LIN {X 0,Y 418.051,Z 411.422,A -85,B 0,C 180,E1 -10031.276,E2 -10031.276} C_VEL
LIN {X 0,Y 417.717,Z 417.579,A -85,B 0,C 180,E1 -10032.621,E2 -10032.621} C_VEL
LIN {X 0,Y 417.509,Z 421.319,A -85,B 0,C 180,E1 -10033.641,E2 -10033.641} C_VEL
LIN {X 0,Y 417.431,Z 423.461,A -85,B 0,C 180,E1 -10034.319,E2 -10034.319} C_VEL
LIN {X 0,Y 417.246,Z 426.661,A -85,B 0,C 180,E1 -10035.665,E2 -10035.665} C_VEL
LIN {X 0,Y 417.136,Z 427.966,A -85,B 0,C 180,E1 -10036.424,E2 -10036.424} C_VEL
LIN {X 0,Y 417.036,Z 429.647,A -85,B 0,C 180,E1 -10037.858,E2 -10037.858} C_VEL
LIN {X 0,Y 417.046,Z 430.141,A -85,B 0,C 180,E1 -10039.316,E2 -10039.316} C_VEL
LIN {X 0,Y 417.093,Z 429.416,A -85,B 0,C 180,E1 -10040.812,E2 -10040.812} C_VEL
LIN {X 0,Y 417.157,Z 428.808,A -85,B 0,C 180,E1 -10041.44,E2 -10041.44} C_VEL
LIN {X 0,Y 417.345,Z 426.876,A -85,B 0,C 180,E1 -10042.684,E2 -10042.684} C_VEL
LIN {X 0,Y 417.561,Z 424.076,A -85,B 0,C 180,E1 -10043.909,E2 -10043.909} C_VEL
LIN {X 0,Y 417.79,Z 420.364,A -85,B 0,C 180,E1 -10045.116,E2 -10045.116} C_VEL
LIN {X 0,Y 418.154,Z 414.507,A -85,B 0,C 180,E1 -10046.541,E2 -10046.541} C_VEL
LIN {X 0,Y 418.405,Z 409.706,A -85,B 0,C 180,E1 -10047.487,E2 -10047.487} C_VEL
LIN {X 0,Y 418.786,Z 403.362,A -85,B 0,C 180,E1 -10048.512,E2 -10048.512} C_VEL
LIN {X 0,Y 419.241,Z 396.766,A -85,B 0,C 180,E1 -10049.391,E2 -10049.391} C_VEL
LIN {X 0,Y 419.666,Z 389.265,A -85,B 0,C 180,E1 -10050.218,E2 -10050.218} C_VEL
LIN {X 0,Y 420.012,Z 381.871,A -85,B 0,C 180,E1 -10050.89,E2 -10050.89} C_VEL
LIN {X 0,Y 420.306,Z 374.017,A -85,B 0,C 180,E1 -10051.473,E2 -10051.473} C_VEL
LIN {X 0,Y 420.619,Z 365.492,A -85,B 0,C 180,E1 -10051.971,E2 -10051.971} C_VEL
LIN {X 0,Y 420.835,Z 356.386,A -85,B 0,C 180,E1 -10052.372,E2 -10052.372} C_VEL
LIN {X 0,Y 420.988,Z 346.253,A -85,B 0,C 180,E1 -10052.673,E2 -10052.673} C_VEL
LIN {X 0,Y 421.787,Z 285.672,A -85,B 0,C 180,E1 -10053.798,E2 -10053.798} C_VEL
LIN {X 0,Y 418.899,Z 271.189,A -85,B 0,C 180,E1 -10054.204,E2 -10054.204} C_VEL
LIN {X 0,Y 418.714,Z 265.669,A -85,B 0,C 180,E1 -10055.455,E2 -10055.455} C_VEL
LIN {X 0,Y 418.251,Z 263.201,A -85,B 0,C 180,E1 -10056.086,E2 -10056.086} C_VEL
LIN {X 0,Y 418.238,Z 263.204,A -85,B 0,C 180,E1 -10059.338,E2 -10059.338} C_VEL
LIN {X 0,Y 418.277,Z 263.2,A -85,B 0,C 180,E1 -10062.397,E2 -10062.397} C_VEL
LIN {X 0,Y 418.292,Z 263.192,A -85,B 0,C 180,E1 -10065.404,E2 -10065.404} C_VEL
LIN {X 0,Y 418.307,Z 263.193,A -85,B 0,C 180,E1 -10068.37,E2 -10068.37} C_VEL
LIN {X 0,Y 418.475,Z 263.171,A -85,B 0,C 180,E1 -10072.28,E2 -10072.28} C_VEL
LIN {X 0,Y 418.521,Z 263.167,A -85,B 0,C 180,E1 -10074.218,E2 -10074.218} C_VEL
LIN {X 0,Y 418.536,Z 263.16,A -85,B 0,C 180,E1 -10078.076,E2 -10078.076} C_VEL
LIN {X 0,Y 418.663,Z 263.146,A -85,B 0,C 180,E1 -10080.001,E2 -10080.001} C_VEL
LIN {X 0,Y 418.503,Z 263.166,A -85,B 0,C 180,E1 -10082.889,E2 -10082.889} C_VEL
LIN {X 0,Y 418.485,Z 263.169,A -85,B 0,C 180,E1 -10086.752,E2 -10086.752} C_VEL
LIN {X 0,Y 418.392,Z 263.179,A -85,B 0,C 180,E1 -10088.696,E2 -10088.696} C_VEL
LIN {X 0,Y 418.307,Z 263.187,A -85,B 0,C 180,E1 -10091.632,E2 -10091.632} C_VEL
LIN {X 0,Y 418.296,Z 263.195,A -85,B 0,C 180,E1 -10094.598,E2 -10094.598} C_VEL
LIN {X 0,Y 418.281,Z 263.188,A -85,B 0,C 180,E1 -10097.605,E2 -10097.605} C_VEL
LIN {X 0,Y 418.243,Z 263.194,A -85,B 0,C 180,E1 -10100.664,E2 -10100.664} C_VEL
LIN {X 0,Y 418.281,Z 263.191,A -85,B 0,C 180,E1 -10103.782,E2 -10103.782} C_VEL
LIN {X 0,Y 418.304,Z 263.19,A -85,B 0,C 180,E1 -10107.072,E2 -10107.072} C_VEL
LIN {X 0,Y 418.255,Z 263.193,A -85,B 0,C 180,E1 -10110.272,E2 -10110.272} C_VEL
LIN {X 0,Y 418.244,Z 263.191,A -85,B 0,C 180,E1 -10113.678,E2 -10113.678} C_VEL
LIN {X 0,Y 418.242,Z 263.193,A -85,B 0,C 180,E1 -10117.224,E2 -10117.224} C_VEL
LIN {X 0,Y 418.261,Z 263.195,A -85,B 0,C 180,E1 -10119.681,E2 -10119.681} C_VEL
LIN {X 0,Y 418.241,Z 263.201,A -85,B 0,C 180,E1 -10122.325,E2 -10122.325} C_VEL
LIN {X 0,Y 418.232,Z 263.199,A -85,B 0,C 180,E1 -10125.11,E2 -10125.11} C_VEL
LIN {X 0,Y 418.237,Z 263.198,A -85,B 0,C 180,E1 -10127.768,E2 -10127.768} C_VEL
LIN {X 0,Y 418.257,Z 263.2,A -85,B 0,C 180,E1 -10130.619,E2 -10130.619} C_VEL
LIN {X 0,Y 418.244,Z 263.199,A -85,B 0,C 180,E1 -10133.977,E2 -10133.977} C_VEL
LIN {X 0,Y 418.256,Z 263.197,A -85,B 0,C 180,E1 -10137.157,E2 -10137.157} C_VEL
LIN {X 0,Y 418.268,Z 263.2,A -85,B 0,C 180,E1 -10140.896,E2 -10140.896} C_VEL
LIN {X 0,Y 418.321,Z 263.192,A -85,B 0,C 180,E1 -10144.1,E2 -10144.1} C_VEL
LIN {X 0,Y 418.342,Z 263.284,A -85,B 0,C 180,E1 -10144.411,E2 -10144.411} C_VEL
LIN {X 0,Y 419.991,Z 273.001,A -85,B 0,C 180,E1 -10146.53,E2 -10146.53} C_VEL
LIN {X 0,Y 419.368,Z 285.804,A -85,B 0,C 180,E1 -10149.139,E2 -10149.139} C_VEL
LIN {X 0,Y 418.6,Z 304.36,A -85,B 0,C 180,E1 -10152.877,E2 -10152.877} C_VEL
LIN {X 0,Y 418.26,Z 314.108,A -85,B 0,C 180,E1 -10154.817,E2 -10154.817} C_VEL
LIN {X 0,Y 421.136,Z 337.432,A -85,B 0,C 180,E1 -10155.378,E2 -10155.378} C_VEL
LIN {X 0,Y 421.116,Z 361.122,A -85,B 0,C 180,E1 -10155.819,E2 -10155.819} C_VEL
LIN {X 0,Y 420.681,Z 393.489,A -85,B 0,C 180,E1 -10156.437,E2 -10156.437} C_VEL
LIN {X 0,Y 420.286,Z 405.245,A -85,B 0,C 180,E1 -10156.831,E2 -10156.831} C_VEL
LIN {X 0,Y 419.731,Z 416.546,A -85,B 0,C 180,E1 -10157.428,E2 -10157.428} C_VEL
LIN {X 0,Y 419.303,Z 425.145,A -85,B 0,C 180,E1 -10158.029,E2 -10158.029} C_VEL
LIN {X 0,Y 418.795,Z 433.417,A -85,B 0,C 180,E1 -10158.751,E2 -10158.751} C_VEL
LIN {X 0,Y 418.4,Z 441.29,A -85,B 0,C 180,E1 -10159.597,E2 -10159.597} C_VEL
LIN {X 0,Y 417.891,Z 450.383,A -85,B 0,C 180,E1 -10160.807,E2 -10160.807} C_VEL
LIN {X 0,Y 417.518,Z 457.415,A -85,B 0,C 180,E1 -10162.018,E2 -10162.018} C_VEL
LIN {X 0,Y 417.309,Z 463.039,A -85,B 0,C 180,E1 -10163.23,E2 -10163.23} C_VEL
LIN {X 0,Y 417.17,Z 468.285,A -85,B 0,C 180,E1 -10164.684,E2 -10164.684} C_VEL
LIN {X 0,Y 417.069,Z 472.133,A -85,B 0,C 180,E1 -10166.135,E2 -10166.135} C_VEL
LIN {X 0,Y 417.133,Z 473.891,A -85,B 0,C 180,E1 -10167.103,E2 -10167.103} C_VEL
LIN {X 0,Y 417.115,Z 475.13,A -85,B 0,C 180,E1 -10168.069,E2 -10168.069} C_VEL
LIN {X 0,Y 417.084,Z 475.881,A -85,B 0,C 180,E1 -10169.035,E2 -10169.035} C_VEL
LIN {X 0,Y 417.112,Z 476.156,A -85,B 0,C 180,E1 -10170,E2 -10170} C_VEL
LIN {X 0,Y 417.095,Z 475.859,A -85,B 0,C 180,E1 -10170.966,E2 -10170.966} C_VEL
LIN {X 0,Y 417.116,Z 474.998,A -85,B 0,C 180,E1 -10171.931,E2 -10171.931} C_VEL
LIN {X 0,Y 417.168,Z 473.644,A -85,B 0,C 180,E1 -10172.897,E2 -10172.897} C_VEL
LIN {X 0,Y 417.102,Z 470.598,A -85,B 0,C 180,E1 -10174.349,E2 -10174.349} C_VEL
LIN {X 0,Y 417.148,Z 466.233,A -85,B 0,C 180,E1 -10175.802,E2 -10175.802} C_VEL
LIN {X 0,Y 417.379,Z 460.161,A -85,B 0,C 180,E1 -10177.255,E2 -10177.255} C_VEL
LIN {X 0,Y 417.559,Z 455.124,A -85,B 0,C 180,E1 -10178.225,E2 -10178.225} C_VEL
LIN {X 0,Y 417.829,Z 449.05,A -85,B 0,C 180,E1 -10179.195,E2 -10179.195} C_VEL
LIN {X 0,Y 418.233,Z 441.657,A -85,B 0,C 180,E1 -10180.163,E2 -10180.163} C_VEL
LIN {X 0,Y 418.592,Z 433.74,A -85,B 0,C 180,E1 -10181.01,E2 -10181.01} C_VEL
LIN {X 0,Y 419.004,Z 425.393,A -85,B 0,C 180,E1 -10181.734,E2 -10181.734} C_VEL
LIN {X 0,Y 419.506,Z 414.774,A -85,B 0,C 180,E1 -10182.456,E2 -10182.456} C_VEL
LIN {X 0,Y 419.974,Z 403.337,A -85,B 0,C 180,E1 -10182.995,E2 -10182.995} C_VEL
LIN {X 0,Y 420.272,Z 393.979,A -85,B 0,C 180,E1 -10183.293,E2 -10183.293} C_VEL
LIN {X 0,Y 420.724,Z 337.989,A -85,B 0,C 180,E1 -10184.335,E2 -10184.335} C_VEL
LIN {X 0,Y 418.181,Z 315.465,A -85,B 0,C 180,E1 -10184.85,E2 -10184.85} C_VEL
LIN {X 0,Y 418.953,Z 297.593,A -85,B 0,C 180,E1 -10188.586,E2 -10188.586} C_VEL
LIN {X 0,Y 419.953,Z 279.654,A -85,B 0,C 180,E1 -10192.378,E2 -10192.378} C_VEL
LIN {X 0,Y 420.149,Z 273.649,A -85,B 0,C 180,E1 -10193.669,E2 -10193.669} C_VEL
LIN {X 0,Y 418.336,Z 263.189,A -85,B 0,C 180,E1 -10196.067,E2 -10196.067} C_VEL
LIN {X 0,Y 418.266,Z 263.197,A -85,B 0,C 180,E1 -10199.161,E2 -10199.161} C_VEL
LIN {X 0,Y 418.258,Z 263.194,A -85,B 0,C 180,E1 -10202.843,E2 -10202.843} C_VEL
LIN {X 0,Y 418.245,Z 263.195,A -85,B 0,C 180,E1 -10206.237,E2 -10206.237} C_VEL
LIN {X 0,Y 418.254,Z 263.199,A -85,B 0,C 180,E1 -10209.681,E2 -10209.681} C_VEL
LIN {X 0,Y 418.229,Z 263.197,A -85,B 0,C 180,E1 -10212.32,E2 -10212.32} C_VEL
LIN {X 0,Y 418.235,Z 263.199,A -85,B 0,C 180,E1 -10215.108,E2 -10215.108} C_VEL
LIN {X 0,Y 418.238,Z 263.2,A -85,B 0,C 180,E1 -10217.766,E2 -10217.766} C_VEL
LIN {X 0,Y 418.243,Z 263.195,A -85,B 0,C 180,E1 -10220.62,E2 -10220.62} C_VEL
LIN {X 0,Y 418.241,Z 263.198,A -85,B 0,C 180,E1 -10223.975,E2 -10223.975} C_VEL
LIN {X 0,Y 418.255,Z 263.196,A -85,B 0,C 180,E1 -10227.155,E2 -10227.155} C_VEL
LIN {X 0,Y 418.266,Z 263.193,A -85,B 0,C 180,E1 -10230.895,E2 -10230.895} C_VEL
LIN {X 0,Y 418.268,Z 263.194,A -85,B 0,C 180,E1 -10234.095,E2 -10234.095} C_VEL
LIN {X 0,Y 418.235,Z 263.2,A -85,B 0,C 180,E1 -10237.263,E2 -10237.263} C_VEL
LIN {X 0,Y 418.279,Z 263.191,A -85,B 0,C 180,E1 -10240.363,E2 -10240.363} C_VEL
LIN {X 0,Y 418.313,Z 263.192,A -85,B 0,C 180,E1 -10243.404,E2 -10243.404} C_VEL
LIN {X 0,Y 418.342,Z 263.184,A -85,B 0,C 180,E1 -10246.999,E2 -10246.999} C_VEL
LIN {X 0,Y 418.336,Z 263.184,A -85,B 0,C 180,E1 -10250.328,E2 -10250.328} C_VEL
LIN {X 0,Y 418.487,Z 263.168,A -85,B 0,C 180,E1 -10253.248,E2 -10253.248} C_VEL
LIN {X 0,Y 418.335,Z 263.186,A -85,B 0,C 180,E1 -10255.181,E2 -10255.181} C_VEL
LIN {X 0,Y 418.539,Z 263.161,A -85,B 0,C 180,E1 -10258.075,E2 -10258.075} C_VEL
LIN {X 0,Y 418.666,Z 263.145,A -85,B 0,C 180,E1 -10259.999,E2 -10259.999} C_VEL
LIN {X 0,Y 418.505,Z 263.163,A -85,B 0,C 180,E1 -10262.887,E2 -10262.887} C_VEL
LIN {X 0,Y 418.487,Z 263.165,A -85,B 0,C 180,E1 -10266.75,E2 -10266.75} C_VEL
LIN {X 0,Y 418.353,Z 263.188,A -85,B 0,C 180,E1 -10269.67,E2 -10269.67} C_VEL
LIN {X 0,Y 418.348,Z 263.184,A -85,B 0,C 180,E1 -10273.005,E2 -10273.005} C_VEL
LIN {X 0,Y 418.305,Z 263.188,A -85,B 0,C 180,E1 -10276.735,E2 -10276.735} C_VEL
LIN {X 0,Y 418.292,Z 263.194,A -85,B 0,C 180,E1 -10279.8,E2 -10279.8} C_VEL
LIN {X 0,Y 418.28,Z 263.196,A -85,B 0,C 180,E1 -10283.78,E2 -10283.78} C_VEL
LIN {X 0,Y 418.302,Z 263.19,A -85,B 0,C 180,E1 -10287.07,E2 -10287.07} C_VEL
LIN {X 0,Y 418.236,Z 263.198,A -85,B 0,C 180,E1 -10290.271,E2 -10290.271} C_VEL
LIN {X 0,Y 418.24,Z 263.203,A -85,B 0,C 180,E1 -10293.677,E2 -10293.677} C_VEL
LIN {X 0,Y 418.238,Z 263.199,A -85,B 0,C 180,E1 -10297.223,E2 -10297.223} C_VEL
LIN {X 0,Y 418.256,Z 263.201,A -85,B 0,C 180,E1 -10299.68,E2 -10299.68} C_VEL
LIN {X 0,Y 418.238,Z 263.197,A -85,B 0,C 180,E1 -10302.323,E2 -10302.323} C_VEL
LIN {X 0,Y 418.252,Z 263.196,A -85,B 0,C 180,E1 -10305.112,E2 -10305.112} C_VEL
LIN {X 0,Y 418.283,Z 263.196,A -85,B 0,C 180,E1 -10307.773,E2 -10307.773} C_VEL
LIN {X 0,Y 418.256,Z 263.2,A -85,B 0,C 180,E1 -10311.559,E2 -10311.559} C_VEL
LIN {X 0,Y 418.25,Z 263.197,A -85,B 0,C 180,E1 -10315.159,E2 -10315.159} C_VEL
LIN {X 0,Y 418.236,Z 263.201,A -85,B 0,C 180,E1 -10317.472,E2 -10317.472} C_VEL
LIN {X 0,Y 418.259,Z 263.194,A -85,B 0,C 180,E1 -10320.895,E2 -10320.895} C_VEL
LIN {X 0,Y 418.262,Z 263.196,A -85,B 0,C 180,E1 -10324.096,E2 -10324.096} C_VEL
LIN {X 0,Y 418.23,Z 263.2,A -85,B 0,C 180,E1 -10327.264,E2 -10327.264} C_VEL
LIN {X 0,Y 418.275,Z 263.193,A -85,B 0,C 180,E1 -10330.364,E2 -10330.364} C_VEL
LIN {X 0,Y 418.308,Z 263.191,A -85,B 0,C 180,E1 -10333.404,E2 -10333.404} C_VEL
LIN {X 0,Y 418.337,Z 263.185,A -85,B 0,C 180,E1 -10336.999,E2 -10336.999} C_VEL
LIN {X 0,Y 418.333,Z 263.186,A -85,B 0,C 180,E1 -10340.328,E2 -10340.328} C_VEL
LIN {X 0,Y 418.504,Z 263.165,A -85,B 0,C 180,E1 -10342.279,E2 -10342.279} C_VEL
LIN {X 0,Y 418.5,Z 263.166,A -85,B 0,C 180,E1 -10344.217,E2 -10344.217} C_VEL
LIN {X 0,Y 418.532,Z 263.163,A -85,B 0,C 180,E1 -10348.075,E2 -10348.075} C_VEL
LIN {X 0,Y 418.662,Z 263.147,A -85,B 0,C 180,E1 -10350,E2 -10350} C_VEL
LIN {X 0,Y 418.491,Z 263.166,A -85,B 0,C 180,E1 -10352.888,E2 -10352.888} C_VEL
LIN {X 0,Y 418.479,Z 263.167,A -85,B 0,C 180,E1 -10356.751,E2 -10356.751} C_VEL
LIN {X 0,Y 418.349,Z 263.189,A -85,B 0,C 180,E1 -10359.671,E2 -10359.671} C_VEL
LIN {X 0,Y 418.323,Z 263.189,A -85,B 0,C 180,E1 -10363.341,E2 -10363.341} C_VEL
LIN {X 0,Y 417.63,Z 263.279,A -85,B 0,C 180,E1 -10364.145,E2 -10364.145} C_VEL
LIN {X 0,Y 414.748,Z 263.635,A -85,B 0,C 180,E1 -10365.45,E2 -10365.45} C_VEL
LIN {X 0,Y 412.33,Z 263.933,A -85,B 0,C 180,E1 -10366.504,E2 -10366.504} C_VEL
LIN {X 0,Y 411.306,Z 264.062,A -85,B 0,C 180,E1 -10367.319,E2 -10367.319} C_VEL
LIN {X 0,Y 411.229,Z 264.071,A -85,B 0,C 180,E1 -10367.595,E2 -10367.595} C_VEL
LIN {X 0,Y 411.186,Z 264.076,A -85,B 0,C 180,E1 -10371.034,E2 -10371.034} C_VEL
LIN {X 0,Y 411.206,Z 264.075,A -85,B 0,C 180,E1 -10374.216,E2 -10374.216} C_VEL
LIN {X 0,Y 411.248,Z 264.071,A -85,B 0,C 180,E1 -10377.478,E2 -10377.478} C_VEL
LIN {X 0,Y 411.181,Z 264.077,A -85,B 0,C 180,E1 -10380.847,E2 -10380.847} C_VEL
LIN {X 0,Y 411.246,Z 264.096,A -85,B 0,C 180,E1 -10382.061,E2 -10382.061} C_VEL
LIN {X 0,Y 411.587,Z 268.326,A -85,B 0,C 180,E1 -10383.21,E2 -10383.21} C_VEL
LIN {X 0,Y 411.503,Z 271.394,A -85,B 0,C 180,E1 -10384.02,E2 -10384.02} C_VEL
LIN {X 0,Y 414.211,Z 286.465,A -85,B 0,C 180,E1 -10384.413,E2 -10384.413} C_VEL
LIN {X 0,Y 413.488,Z 348.411,A -85,B 0,C 180,E1 -10385.58,E2 -10385.58} C_VEL
LIN {X 0,Y 413.271,Z 359.308,A -85,B 0,C 180,E1 -10385.945,E2 -10385.945} C_VEL
LIN {X 0,Y 412.974,Z 371.003,A -85,B 0,C 180,E1 -10386.556,E2 -10386.556} C_VEL
LIN {X 0,Y 412.627,Z 379.505,A -85,B 0,C 180,E1 -10387.152,E2 -10387.152} C_VEL
LIN {X 0,Y 412.312,Z 387.5,A -85,B 0,C 180,E1 -10387.851,E2 -10387.851} C_VEL
LIN {X 0,Y 412.044,Z 393.555,A -85,B 0,C 180,E1 -10388.48,E2 -10388.48} C_VEL
LIN {X 0,Y 411.548,Z 401.376,A -85,B 0,C 180,E1 -10389.468,E2 -10389.468} C_VEL
LIN {X 0,Y 411.217,Z 408.029,A -85,B 0,C 180,E1 -10390.499,E2 -10390.499} C_VEL
LIN {X 0,Y 410.792,Z 415.077,A -85,B 0,C 180,E1 -10391.852,E2 -10391.852} C_VEL
LIN {X 0,Y 410.531,Z 420.558,A -85,B 0,C 180,E1 -10393.216,E2 -10393.216} C_VEL
LIN {X 0,Y 410.322,Z 424.691,A -85,B 0,C 180,E1 -10394.606,E2 -10394.606} C_VEL
LIN {X 0,Y 410.204,Z 426.537,A -85,B 0,C 180,E1 -10395.378,E2 -10395.378} C_VEL
LIN {X 0,Y 410.015,Z 428.851,A -85,B 0,C 180,E1 -10396.716,E2 -10396.716} C_VEL
LIN {X 0,Y 409.94,Z 430.159,A -85,B 0,C 180,E1 -10398.041,E2 -10398.041} C_VEL
LIN {X 0,Y 409.958,Z 430.536,A -85,B 0,C 180,E1 -10399.351,E2 -10399.351} C_VEL
LIN {X 0,Y 410.015,Z 430.031,A -85,B 0,C 180,E1 -10400.64,E2 -10400.64} C_VEL
LIN {X 0,Y 410.157,Z 428.502,A -85,B 0,C 180,E1 -10402.016,E2 -10402.016} C_VEL
LIN {X 0,Y 410.406,Z 425.467,A -85,B 0,C 180,E1 -10403.594,E2 -10403.594} C_VEL
LIN {X 0,Y 410.646,Z 422,A -85,B 0,C 180,E1 -10404.85,E2 -10404.85} C_VEL
LIN {X 0,Y 411.005,Z 416.954,A -85,B 0,C 180,E1 -10406.24,E2 -10406.24} C_VEL
LIN {X 0,Y 411.346,Z 411.241,A -85,B 0,C 180,E1 -10407.455,E2 -10407.455} C_VEL
LIN {X 0,Y 411.763,Z 404.558,A -85,B 0,C 180,E1 -10408.581,E2 -10408.581} C_VEL
LIN {X 0,Y 412.277,Z 397.73,A -85,B 0,C 180,E1 -10409.521,E2 -10409.521} C_VEL
LIN {X 0,Y 412.744,Z 389.869,A -85,B 0,C 180,E1 -10410.411,E2 -10410.411} C_VEL
LIN {X 0,Y 413.145,Z 381.963,A -85,B 0,C 180,E1 -10411.14,E2 -10411.14} C_VEL
LIN {X 0,Y 413.474,Z 373.168,A -85,B 0,C 180,E1 -10411.792,E2 -10411.792} C_VEL
LIN {X 0,Y 413.87,Z 363.339,A -85,B 0,C 180,E1 -10412.347,E2 -10412.347} C_VEL
LIN {X 0,Y 414.112,Z 351.983,A -85,B 0,C 180,E1 -10412.797,E2 -10412.797} C_VEL
LIN {X 0,Y 414.341,Z 333.574,A -85,B 0,C 180,E1 -10413.188,E2 -10413.188} C_VEL
LIN {X 0,Y 414.953,Z 286.313,A -85,B 0,C 180,E1 -10414.077,E2 -10414.077} C_VEL
LIN {X 0,Y 411.987,Z 271.478,A -85,B 0,C 180,E1 -10414.524,E2 -10414.524} C_VEL
LIN {X 0,Y 411.782,Z 267.012,A -85,B 0,C 180,E1 -10415.552,E2 -10415.552} C_VEL
LIN {X 0,Y 411.209,Z 264.079,A -85,B 0,C 180,E1 -10416.32,E2 -10416.32} C_VEL
LIN {X 0,Y 411.22,Z 264.08,A -85,B 0,C 180,E1 -10420.014,E2 -10420.014} C_VEL
LIN {X 0,Y 411.252,Z 264.07,A -85,B 0,C 180,E1 -10423.132,E2 -10423.132} C_VEL
LIN {X 0,Y 411.295,Z 264.066,A -85,B 0,C 180,E1 -10426.897,E2 -10426.897} C_VEL
LIN {X 0,Y 411.284,Z 264.067,A -85,B 0,C 180,E1 -10430.162,E2 -10430.162} C_VEL
LIN {X 0,Y 411.447,Z 264.045,A -85,B 0,C 180,E1 -10433.134,E2 -10433.134} C_VEL
LIN {X 0,Y 411.307,Z 264.061,A -85,B 0,C 180,E1 -10435.1,E2 -10435.1} C_VEL
LIN {X 0,Y 411.505,Z 264.035,A -85,B 0,C 180,E1 -10438.043,E2 -10438.043} C_VEL
LIN {X 0,Y 411.633,Z 264.022,A -85,B 0,C 180,E1 -10440.001,E2 -10440.001} C_VEL
LIN {X 0,Y 411.458,Z 264.043,A -85,B 0,C 180,E1 -10442.938,E2 -10442.938} C_VEL
LIN {X 0,Y 411.452,Z 264.043,A -85,B 0,C 180,E1 -10446.868,E2 -10446.868} C_VEL
LIN {X 0,Y 411.346,Z 264.057,A -85,B 0,C 180,E1 -10448.846,E2 -10448.846} C_VEL
LIN {X 0,Y 411.276,Z 264.063,A -85,B 0,C 180,E1 -10451.834,E2 -10451.834} C_VEL
LIN {X 0,Y 411.253,Z 264.069,A -85,B 0,C 180,E1 -10454.854,E2 -10454.854} C_VEL
LIN {X 0,Y 411.246,Z 264.066,A -85,B 0,C 180,E1 -10457.916,E2 -10457.916} C_VEL
LIN {X 0,Y 411.189,Z 264.071,A -85,B 0,C 180,E1 -10461.035,E2 -10461.035} C_VEL
LIN {X 0,Y 411.221,Z 264.074,A -85,B 0,C 180,E1 -10464.216,E2 -10464.216} C_VEL
LIN {X 0,Y 411.254,Z 264.067,A -85,B 0,C 180,E1 -10467.479,E2 -10467.479} C_VEL
LIN {X 0,Y 411.193,Z 264.078,A -85,B 0,C 180,E1 -10470.848,E2 -10470.848} C_VEL
LIN {X 0,Y 411.201,Z 264.073,A -85,B 0,C 180,E1 -10474.335,E2 -10474.335} C_VEL
LIN {X 0,Y 411.2,Z 264.072,A -85,B 0,C 180,E1 -10477.974,E2 -10477.974} C_VEL
LIN {X 0,Y 411.196,Z 264.074,A -85,B 0,C 180,E1 -10481.235,E2 -10481.235} C_VEL
LIN {X 0,Y 411.172,Z 264.08,A -85,B 0,C 180,E1 -10484.491,E2 -10484.491} C_VEL
LIN {X 0,Y 411.175,Z 264.081,A -85,B 0,C 180,E1 -10488.196,E2 -10488.196} C_VEL
LIN {X 0,Y 411.221,Z 264.075,A -85,B 0,C 180,E1 -10490.778,E2 -10490.778} C_VEL
LIN {X 0,Y 411.198,Z 264.081,A -85,B 0,C 180,E1 -10494.472,E2 -10494.472} C_VEL
LIN {X 0,Y 411.206,Z 264.078,A -85,B 0,C 180,E1 -10496.874,E2 -10496.874} C_VEL
LIN {X 0,Y 411.232,Z 264.078,A -85,B 0,C 180,E1 -10500.645,E2 -10500.645} C_VEL
LIN {X 0,Y 411.298,Z 264.122,A -85,B 0,C 180,E1 -10504.186,E2 -10504.186} C_VEL
LIN {X 0,Y 413.046,Z 274.182,A -85,B 0,C 180,E1 -10506.414,E2 -10506.414} C_VEL
LIN {X 0,Y 412.38,Z 286.777,A -85,B 0,C 180,E1 -10509.03,E2 -10509.03} C_VEL
LIN {X 0,Y 411.623,Z 304.5,A -85,B 0,C 180,E1 -10512.667,E2 -10512.667} C_VEL
LIN {X 0,Y 411.25,Z 313.796,A -85,B 0,C 180,E1 -10514.517,E2 -10514.517} C_VEL
LIN {X 0,Y 413.92,Z 333.925,A -85,B 0,C 180,E1 -10515.022,E2 -10515.022} C_VEL
LIN {X 0,Y 414.495,Z 343.91,A -85,B 0,C 180,E1 -10515.24,E2 -10515.24} C_VEL
LIN {X 0,Y 413.864,Z 392.496,A -85,B 0,C 180,E1 -10516.171,E2 -10516.171} C_VEL
LIN {X 0,Y 413.499,Z 403.048,A -85,B 0,C 180,E1 -10516.517,E2 -10516.517} C_VEL
LIN {X 0,Y 412.933,Z 414.579,A -85,B 0,C 180,E1 -10517.093,E2 -10517.093} C_VEL
LIN {X 0,Y 412.397,Z 423.48,A -85,B 0,C 180,E1 -10517.701,E2 -10517.701} C_VEL
LIN {X 0,Y 411.919,Z 431.978,A -85,B 0,C 180,E1 -10518.436,E2 -10518.436} C_VEL
LIN {X 0,Y 411.467,Z 440.025,A -85,B 0,C 180,E1 -10519.296,E2 -10519.296} C_VEL
LIN {X 0,Y 411.039,Z 446.688,A -85,B 0,C 180,E1 -10520.156,E2 -10520.156} C_VEL
LIN {X 0,Y 410.644,Z 453.035,A -85,B 0,C 180,E1 -10521.14,E2 -10521.14} C_VEL
LIN {X 0,Y 410.41,Z 458.316,A -85,B 0,C 180,E1 -10522.126,E2 -10522.126} C_VEL
LIN {X 0,Y 410.254,Z 462.724,A -85,B 0,C 180,E1 -10523.113,E2 -10523.113} C_VEL
LIN {X 0,Y 410.067,Z 466.387,A -85,B 0,C 180,E1 -10524.098,E2 -10524.098} C_VEL
LIN {X 0,Y 410.074,Z 469.408,A -85,B 0,C 180,E1 -10525.085,E2 -10525.085} C_VEL
LIN {X 0,Y 409.985,Z 471.787,A -85,B 0,C 180,E1 -10526.069,E2 -10526.069} C_VEL
LIN {X 0,Y 410.031,Z 473.534,A -85,B 0,C 180,E1 -10527.053,E2 -10527.053} C_VEL
LIN {X 0,Y 410.042,Z 474.758,A -85,B 0,C 180,E1 -10528.036,E2 -10528.036} C_VEL
LIN {X 0,Y 410.005,Z 475.493,A -85,B 0,C 180,E1 -10529.018,E2 -10529.018} C_VEL
LIN {X 0,Y 410.028,Z 475.753,A -85,B 0,C 180,E1 -10530,E2 -10530} C_VEL
LIN {X 0,Y 410.015,Z 475.455,A -85,B 0,C 180,E1 -10530.982,E2 -10530.982} C_VEL
LIN {X 0,Y 410.044,Z 474.578,A -85,B 0,C 180,E1 -10531.965,E2 -10531.965} C_VEL
LIN {X 0,Y 410.066,Z 473.204,A -85,B 0,C 180,E1 -10532.947,E2 -10532.947} C_VEL
LIN {X 0,Y 410.031,Z 470.137,A -85,B 0,C 180,E1 -10534.424,E2 -10534.424} C_VEL
LIN {X 0,Y 410.057,Z 465.735,A -85,B 0,C 180,E1 -10535.903,E2 -10535.903} C_VEL
LIN {X 0,Y 410.278,Z 460.805,A -85,B 0,C 180,E1 -10537.134,E2 -10537.134} C_VEL
LIN {X 0,Y 410.494,Z 454.54,A -85,B 0,C 180,E1 -10538.368,E2 -10538.368} C_VEL
LIN {X 0,Y 410.776,Z 448.421,A -85,B 0,C 180,E1 -10539.354,E2 -10539.354} C_VEL
LIN {X 0,Y 411.239,Z 440.982,A -85,B 0,C 180,E1 -10540.337,E2 -10540.337} C_VEL
LIN {X 0,Y 411.626,Z 433.005,A -85,B 0,C 180,E1 -10541.199,E2 -10541.199} C_VEL
LIN {X 0,Y 412.123,Z 423.07,A -85,B 0,C 180,E1 -10542.058,E2 -10542.058} C_VEL
LIN {X 0,Y 412.632,Z 411.402,A -85,B 0,C 180,E1 -10542.792,E2 -10542.792} C_VEL
LIN {X 0,Y 413.038,Z 402.017,A -85,B 0,C 180,E1 -10543.217,E2 -10543.217} C_VEL
LIN {X 0,Y 413.315,Z 393.423,A -85,B 0,C 180,E1 -10543.49,E2 -10543.49} C_VEL
LIN {X 0,Y 413.819,Z 338.887,A -85,B 0,C 180,E1 -10544.522,E2 -10544.522} C_VEL
LIN {X 0,Y 411.133,Z 315.102,A -85,B 0,C 180,E1 -10545.079,E2 -10545.079} C_VEL
LIN {X 0,Y 411.918,Z 298.292,A -85,B 0,C 180,E1 -10548.657,E2 -10548.657} C_VEL
LIN {X 0,Y 412.973,Z 280.369,A -85,B 0,C 180,E1 -10552.514,E2 -10552.514} C_VEL
LIN {X 0,Y 413.071,Z 274.195,A -85,B 0,C 180,E1 -10553.866,E2 -10553.866} C_VEL
LIN {X 0,Y 411.288,Z 264.066,A -85,B 0,C 180,E1 -10556.24,E2 -10556.24} C_VEL
LIN {X 0,Y 411.201,Z 264.077,A -85,B 0,C 180,E1 -10559.712,E2 -10559.712} C_VEL
LIN {X 0,Y 411.207,Z 264.074,A -85,B 0,C 180,E1 -10563.155,E2 -10563.155} C_VEL
LIN {X 0,Y 411.193,Z 264.073,A -85,B 0,C 180,E1 -10566.552,E2 -10566.552} C_VEL
LIN {X 0,Y 411.217,Z 264.075,A -85,B 0,C 180,E1 -10569.728,E2 -10569.728} C_VEL
LIN {X 0,Y 411.173,Z 264.078,A -85,B 0,C 180,E1 -10573.133,E2 -10573.133} C_VEL
LIN {X 0,Y 411.166,Z 264.08,A -85,B 0,C 180,E1 -10575.88,E2 -10575.88} C_VEL
LIN {X 0,Y 411.162,Z 264.078,A -85,B 0,C 180,E1 -10578.771,E2 -10578.771} C_VEL
LIN {X 0,Y 411.19,Z 264.076,A -85,B 0,C 180,E1 -10582.025,E2 -10582.025} C_VEL
LIN {X 0,Y 411.204,Z 264.078,A -85,B 0,C 180,E1 -10585.666,E2 -10585.666} C_VEL
LIN {X 0,Y 411.187,Z 264.077,A -85,B 0,C 180,E1 -10589.152,E2 -10589.152} C_VEL
LIN {X 0,Y 411.256,Z 264.066,A -85,B 0,C 180,E1 -10592.522,E2 -10592.522} C_VEL
LIN {X 0,Y 411.224,Z 264.074,A -85,B 0,C 180,E1 -10595.784,E2 -10595.784} C_VEL
LIN {X 0,Y 411.193,Z 264.075,A -85,B 0,C 180,E1 -10598.965,E2 -10598.965} C_VEL
LIN {X 0,Y 411.248,Z 264.068,A -85,B 0,C 180,E1 -10602.084,E2 -10602.084} C_VEL
LIN {X 0,Y 411.255,Z 264.068,A -85,B 0,C 180,E1 -10605.146,E2 -10605.146} C_VEL
LIN {X 0,Y 411.279,Z 264.064,A -85,B 0,C 180,E1 -10608.166,E2 -10608.166} C_VEL
LIN {X 0,Y 411.436,Z 264.045,A -85,B 0,C 180,E1 -10612.188,E2 -10612.188} C_VEL
LIN {X 0,Y 411.469,Z 264.041,A -85,B 0,C 180,E1 -10614.117,E2 -10614.117} C_VEL
LIN {X 0,Y 411.508,Z 264.037,A -85,B 0,C 180,E1 -10618.042,E2 -10618.042} C_VEL
LIN {X 0,Y 411.636,Z 264.021,A -85,B 0,C 180,E1 -10619.999,E2 -10619.999} C_VEL
LIN {X 0,Y 411.46,Z 264.041,A -85,B 0,C 180,E1 -10622.936,E2 -10622.936} C_VEL
LIN {X 0,Y 411.454,Z 264.042,A -85,B 0,C 180,E1 -10626.866,E2 -10626.866} C_VEL
LIN {X 0,Y 411.301,Z 264.065,A -85,B 0,C 180,E1 -10629.838,E2 -10629.838} C_VEL
LIN {X 0,Y 411.306,Z 264.061,A -85,B 0,C 180,E1 -10633.108,E2 -10633.108} C_VEL
LIN {X 0,Y 411.25,Z 264.067,A -85,B 0,C 180,E1 -10636.888,E2 -10636.888} C_VEL
LIN {X 0,Y 411.247,Z 264.07,A -85,B 0,C 180,E1 -10639.985,E2 -10639.985} C_VEL
LIN {X 0,Y 411.195,Z 264.075,A -85,B 0,C 180,E1 -10643.147,E2 -10643.147} C_VEL
LIN {X 0,Y 411.23,Z 264.07,A -85,B 0,C 180,E1 -10646.38,E2 -10646.38} C_VEL
LIN {X 0,Y 411.192,Z 264.08,A -85,B 0,C 180,E1 -10649.712,E2 -10649.712} C_VEL
LIN {X 0,Y 411.198,Z 264.075,A -85,B 0,C 180,E1 -10653.155,E2 -10653.155} C_VEL
LIN {X 0,Y 411.187,Z 264.075,A -85,B 0,C 180,E1 -10656.553,E2 -10656.553} C_VEL
LIN {X 0,Y 411.219,Z 264.077,A -85,B 0,C 180,E1 -10659.73,E2 -10659.73} C_VEL
LIN {X 0,Y 411.173,Z 264.078,A -85,B 0,C 180,E1 -10663.132,E2 -10663.132} C_VEL
LIN {X 0,Y 411.219,Z 264.075,A -85,B 0,C 180,E1 -10665.872,E2 -10665.872} C_VEL
LIN {X 0,Y 411.201,Z 264.073,A -85,B 0,C 180,E1 -10668.764,E2 -10668.764} C_VEL
LIN {X 0,Y 411.194,Z 264.077,A -85,B 0,C 180,E1 -10672.027,E2 -10672.027} C_VEL
LIN {X 0,Y 411.197,Z 264.08,A -85,B 0,C 180,E1 -10675.666,E2 -10675.666} C_VEL
LIN {X 0,Y 411.18,Z 264.077,A -85,B 0,C 180,E1 -10679.152,E2 -10679.152} C_VEL
LIN {X 0,Y 411.25,Z 264.068,A -85,B 0,C 180,E1 -10682.522,E2 -10682.522} C_VEL
LIN {X 0,Y 411.219,Z 264.076,A -85,B 0,C 180,E1 -10685.784,E2 -10685.784} C_VEL
LIN {X 0,Y 411.19,Z 264.075,A -85,B 0,C 180,E1 -10688.966,E2 -10688.966} C_VEL
LIN {X 0,Y 411.244,Z 264.07,A -85,B 0,C 180,E1 -10692.085,E2 -10692.085} C_VEL
LIN {X 0,Y 411.251,Z 264.068,A -85,B 0,C 180,E1 -10695.147,E2 -10695.147} C_VEL
LIN {X 0,Y 411.276,Z 264.066,A -85,B 0,C 180,E1 -10698.167,E2 -10698.167} C_VEL
LIN {X 0,Y 411.473,Z 264.041,A -85,B 0,C 180,E1 -10702.146,E2 -10702.146} C_VEL
LIN {X 0,Y 411.462,Z 264.043,A -85,B 0,C 180,E1 -10704.118,E2 -10704.118} C_VEL
LIN {X 0,Y 411.501,Z 264.039,A -85,B 0,C 180,E1 -10708.042,E2 -10708.042} C_VEL
LIN {X 0,Y 411.632,Z 264.023,A -85,B 0,C 180,E1 -10710,E2 -10710} C_VEL
LIN {X 0,Y 411.448,Z 264.043,A -85,B 0,C 180,E1 -10712.937,E2 -10712.937} C_VEL
LIN {X 0,Y 411.443,Z 264.043,A -85,B 0,C 180,E1 -10716.867,E2 -10716.867} C_VEL
LIN {X 0,Y 411.297,Z 264.066,A -85,B 0,C 180,E1 -10719.838,E2 -10719.838} C_VEL
LIN {X 0,Y 411.282,Z 264.065,A -85,B 0,C 180,E1 -10723.33,E2 -10723.33} C_VEL
LIN {X 0,Y 411.247,Z 264.068,A -85,B 0,C 180,E1 -10726.889,E2 -10726.889} C_VEL
LIN {X 0,Y 411.229,Z 264.071,A -85,B 0,C 180,E1 -10727.595,E2 -10727.595} C_VEL
LIN {X 0,Y 410.569,Z 264.157,A -85,B 0,C 180,E1 -10728.412,E2 -10728.412} C_VEL
LIN {X 0,Y 407.681,Z 264.518,A -85,B 0,C 180,E1 -10729.741,E2 -10729.741} C_VEL
LIN {X 0,Y 405.237,Z 264.82,A -85,B 0,C 180,E1 -10730.813,E2 -10730.813} C_VEL
LIN {X 0,Y 404.201,Z 264.95,A -85,B 0,C 180,E1 -10731.643,E2 -10731.643} C_VEL
LIN {X 0,Y 404.125,Z 264.955,A -85,B 0,C 180,E1 -10731.925,E2 -10731.925} C_VEL
LIN {X 0,Y 404.204,Z 264.947,A -85,B 0,C 180,E1 -10735.296,E2 -10735.296} C_VEL
LIN {X 0,Y 404.184,Z 264.951,A -85,B 0,C 180,E1 -10738,E2 -10738} C_VEL
LIN {X 0,Y 404.181,Z 264.954,A -85,B 0,C 180,E1 -10741.932,E2 -10741.932} C_VEL
LIN {X 0,Y 404.593,Z 268.92,A -85,B 0,C 180,E1 -10743.035,E2 -10743.035} C_VEL
LIN {X 0,Y 404.505,Z 271.699,A -85,B 0,C 180,E1 -10743.777,E2 -10743.777} C_VEL
LIN {X 0,Y 407.254,Z 286.825,A -85,B 0,C 180,E1 -10744.188,E2 -10744.188} C_VEL
LIN {X 0,Y 406.568,Z 348.665,A -85,B 0,C 180,E1 -10745.379,E2 -10745.379} C_VEL
LIN {X 0,Y 406.32,Z 359.631,A -85,B 0,C 180,E1 -10745.75,E2 -10745.75} C_VEL
LIN {X 0,Y 406.018,Z 371.146,A -85,B 0,C 180,E1 -10746.359,E2 -10746.359} C_VEL
LIN {X 0,Y 405.633,Z 380.343,A -85,B 0,C 180,E1 -10747.018,E2 -10747.018} C_VEL
LIN {X 0,Y 405.289,Z 389.311,A -85,B 0,C 180,E1 -10747.837,E2 -10747.837} C_VEL
LIN {X 0,Y 404.85,Z 396.796,A -85,B 0,C 180,E1 -10748.677,E2 -10748.677} C_VEL
LIN {X 0,Y 404.393,Z 404.219,A -85,B 0,C 180,E1 -10749.692,E2 -10749.692} C_VEL
LIN {X 0,Y 403.997,Z 412.073,A -85,B 0,C 180,E1 -10751.047,E2 -10751.047} C_VEL
LIN {X 0,Y 403.632,Z 417.096,A -85,B 0,C 180,E1 -10752.136,E2 -10752.136} C_VEL
LIN {X 0,Y 403.507,Z 420.391,A -85,B 0,C 180,E1 -10752.987,E2 -10752.987} C_VEL
LIN {X 0,Y 403.277,Z 424.701,A -85,B 0,C 180,E1 -10754.398,E2 -10754.398} C_VEL
LIN {X 0,Y 403.053,Z 427.723,A -85,B 0,C 180,E1 -10755.777,E2 -10755.777} C_VEL
LIN {X 0,Y 402.892,Z 429.695,A -85,B 0,C 180,E1 -10757.134,E2 -10757.134} C_VEL
LIN {X 0,Y 402.855,Z 430.755,A -85,B 0,C 180,E1 -10758.602,E2 -10758.602} C_VEL
LIN {X 0,Y 402.897,Z 430.72,A -85,B 0,C 180,E1 -10760.13,E2 -10760.13} C_VEL
LIN {X 0,Y 403.046,Z 429.494,A -85,B 0,C 180,E1 -10761.689,E2 -10761.689} C_VEL
LIN {X 0,Y 403.345,Z 425.933,A -85,B 0,C 180,E1 -10763.672,E2 -10763.672} C_VEL
LIN {X 0,Y 403.594,Z 422.561,A -85,B 0,C 180,E1 -10764.927,E2 -10764.927} C_VEL
LIN {X 0,Y 403.919,Z 418.22,A -85,B 0,C 180,E1 -10766.168,E2 -10766.168} C_VEL
LIN {X 0,Y 404.377,Z 411.546,A -85,B 0,C 180,E1 -10767.65,E2 -10767.65} C_VEL
LIN {X 0,Y 404.898,Z 404.056,A -85,B 0,C 180,E1 -10768.911,E2 -10768.911} C_VEL
LIN {X 0,Y 405.393,Z 397.449,A -85,B 0,C 180,E1 -10769.819,E2 -10769.819} C_VEL
LIN {X 0,Y 405.892,Z 389.506,A -85,B 0,C 180,E1 -10770.717,E2 -10770.717} C_VEL
LIN {X 0,Y 406.33,Z 381.08,A -85,B 0,C 180,E1 -10771.488,E2 -10771.488} C_VEL
LIN {X 0,Y 406.732,Z 371.348,A -85,B 0,C 180,E1 -10772.191,E2 -10772.191} C_VEL
LIN {X 0,Y 407.099,Z 359.21,A -85,B 0,C 180,E1 -10772.811,E2 -10772.811} C_VEL
LIN {X 0,Y 407.327,Z 349.398,A -85,B 0,C 180,E1 -10773.14,E2 -10773.14} C_VEL
LIN {X 0,Y 408.127,Z 286.706,A -85,B 0,C 180,E1 -10774.37,E2 -10774.37} C_VEL
LIN {X 0,Y 405.072,Z 271.868,A -85,B 0,C 180,E1 -10774.844,E2 -10774.844} C_VEL
LIN {X 0,Y 404.648,Z 267.381,A -85,B 0,C 180,E1 -10775.912,E2 -10775.912} C_VEL
LIN {X 0,Y 404.159,Z 264.957,A -85,B 0,C 180,E1 -10776.533,E2 -10776.533} C_VEL
LIN {X 0,Y 404.18,Z 264.956,A -85,B 0,C 180,E1 -10779.875,E2 -10779.875} C_VEL
LIN {X 0,Y 404.205,Z 264.949,A -85,B 0,C 180,E1 -10782.994,E2 -10782.994} C_VEL
LIN {X 0,Y 404.272,Z 264.94,A -85,B 0,C 180,E1 -10786.94,E2 -10786.94} C_VEL
LIN {X 0,Y 404.249,Z 264.943,A -85,B 0,C 180,E1 -10789.989,E2 -10789.989} C_VEL
LIN {X 0,Y 404.394,Z 264.925,A -85,B 0,C 180,E1 -10793.013,E2 -10793.013} C_VEL
LIN {X 0,Y 404.279,Z 264.937,A -85,B 0,C 180,E1 -10795.014,E2 -10795.014} C_VEL
LIN {X 0,Y 404.474,Z 264.911,A -85,B 0,C 180,E1 -10798.009,E2 -10798.009} C_VEL
LIN {X 0,Y 404.602,Z 264.898,A -85,B 0,C 180,E1 -10800.001,E2 -10800.001} C_VEL
LIN {X 0,Y 404.415,Z 264.92,A -85,B 0,C 180,E1 -10802.989,E2 -10802.989} C_VEL
LIN {X 0,Y 404.403,Z 264.921,A -85,B 0,C 180,E1 -10806.988,E2 -10806.988} C_VEL
LIN {X 0,Y 404.25,Z 264.94,A -85,B 0,C 180,E1 -10810.013,E2 -10810.013} C_VEL
LIN {X 0,Y 404.259,Z 264.937,A -85,B 0,C 180,E1 -10813.212,E2 -10813.212} C_VEL
LIN {X 0,Y 404.209,Z 264.943,A -85,B 0,C 180,E1 -10817.008,E2 -10817.008} C_VEL
LIN {X 0,Y 404.157,Z 264.95,A -85,B 0,C 180,E1 -10820.353,E2 -10820.353} C_VEL
LIN {X 0,Y 404.163,Z 264.949,A -85,B 0,C 180,E1 -10823.576,E2 -10823.576} C_VEL
LIN {X 0,Y 404.178,Z 264.943,A -85,B 0,C 180,E1 -10825.767,E2 -10825.767} C_VEL
LIN {X 0,Y 404.193,Z 264.948,A -85,B 0,C 180,E1 -10828,E2 -10828} C_VEL
LIN {X 0,Y 404.137,Z 264.954,A -85,B 0,C 180,E1 -10831.56,E2 -10831.56} C_VEL
LIN {X 0,Y 404.181,Z 264.95,A -85,B 0,C 180,E1 -10835.017,E2 -10835.017} C_VEL
LIN {X 0,Y 404.159,Z 264.955,A -85,B 0,C 180,E1 -10838.757,E2 -10838.757} C_VEL
LIN {X 0,Y 404.146,Z 264.952,A -85,B 0,C 180,E1 -10841.605,E2 -10841.605} C_VEL
LIN {X 0,Y 404.142,Z 264.956,A -85,B 0,C 180,E1 -10844.523,E2 -10844.523} C_VEL
LIN {X 0,Y 404.133,Z 264.955,A -85,B 0,C 180,E1 -10847.297,E2 -10847.297} C_VEL
LIN {X 0,Y 404.167,Z 264.952,A -85,B 0,C 180,E1 -10849.956,E2 -10849.956} C_VEL
LIN {X 0,Y 404.138,Z 264.955,A -85,B 0,C 180,E1 -10853.125,E2 -10853.125} C_VEL
LIN {X 0,Y 404.144,Z 264.958,A -85,B 0,C 180,E1 -10856.189,E2 -10856.189} C_VEL
LIN {X 0,Y 404.145,Z 264.957,A -85,B 0,C 180,E1 -10859.716,E2 -10859.716} C_VEL
LIN {X 0,Y 404.207,Z 264.95,A -85,B 0,C 180,E1 -10863.125,E2 -10863.125} C_VEL
LIN {X 0,Y 404.269,Z 265.059,A -85,B 0,C 180,E1 -10863.963,E2 -10863.963} C_VEL
LIN {X 0,Y 406.073,Z 275.36,A -85,B 0,C 180,E1 -10866.3,E2 -10866.3} C_VEL
LIN {X 0,Y 405.381,Z 288.811,A -85,B 0,C 180,E1 -10869.135,E2 -10869.135} C_VEL
LIN {X 0,Y 404.513,Z 306.663,A -85,B 0,C 180,E1 -10872.857,E2 -10872.857} C_VEL
LIN {X 0,Y 404.285,Z 313.022,A -85,B 0,C 180,E1 -10874.175,E2 -10874.175} C_VEL
LIN {X 0,Y 407.161,Z 334.798,A -85,B 0,C 180,E1 -10874.756,E2 -10874.756} C_VEL
LIN {X 0,Y 407.694,Z 343.502,A -85,B 0,C 180,E1 -10874.951,E2 -10874.951} C_VEL
LIN {X 0,Y 407.074,Z 391.818,A -85,B 0,C 180,E1 -10875.896,E2 -10875.896} C_VEL
LIN {X 0,Y 406.692,Z 401.832,A -85,B 0,C 180,E1 -10876.223,E2 -10876.223} C_VEL
LIN {X 0,Y 406.157,Z 412.659,A -85,B 0,C 180,E1 -10876.746,E2 -10876.746} C_VEL
LIN {X 0,Y 405.469,Z 423.414,A -85,B 0,C 180,E1 -10877.487,E2 -10877.487} C_VEL
LIN {X 0,Y 404.965,Z 431.836,A -85,B 0,C 180,E1 -10878.234,E2 -10878.234} C_VEL
LIN {X 0,Y 404.482,Z 439.825,A -85,B 0,C 180,E1 -10879.109,E2 -10879.109} C_VEL
LIN {X 0,Y 404.02,Z 446.445,A -85,B 0,C 180,E1 -10879.983,E2 -10879.983} C_VEL
LIN {X 0,Y 403.616,Z 452.759,A -85,B 0,C 180,E1 -10880.984,E2 -10880.984} C_VEL
LIN {X 0,Y 403.361,Z 458.022,A -85,B 0,C 180,E1 -10881.988,E2 -10881.988} C_VEL
LIN {X 0,Y 403.19,Z 462.412,A -85,B 0,C 180,E1 -10882.992,E2 -10882.992} C_VEL
LIN {X 0,Y 402.987,Z 466.057,A -85,B 0,C 180,E1 -10883.994,E2 -10883.994} C_VEL
LIN {X 0,Y 402.959,Z 470.262,A -85,B 0,C 180,E1 -10885.499,E2 -10885.499} C_VEL
LIN {X 0,Y 402.929,Z 473.178,A -85,B 0,C 180,E1 -10887.001,E2 -10887.001} C_VEL
LIN {X 0,Y 402.971,Z 474.389,A -85,B 0,C 180,E1 -10888.001,E2 -10888.001} C_VEL
LIN {X 0,Y 402.929,Z 475.106,A -85,B 0,C 180,E1 -10889.001,E2 -10889.001} C_VEL
LIN {X 0,Y 402.948,Z 475.349,A -85,B 0,C 180,E1 -10890,E2 -10890} C_VEL
LIN {X 0,Y 402.938,Z 475.049,A -85,B 0,C 180,E1 -10891,E2 -10891} C_VEL
LIN {X 0,Y 402.974,Z 474.157,A -85,B 0,C 180,E1 -10891.999,E2 -10891.999} C_VEL
LIN {X 0,Y 402.965,Z 472.76,A -85,B 0,C 180,E1 -10892.999,E2 -10892.999} C_VEL
LIN {X 0,Y 402.962,Z 469.672,A -85,B 0,C 180,E1 -10894.502,E2 -10894.502} C_VEL
LIN {X 0,Y 402.987,Z 465.229,A -85,B 0,C 180,E1 -10896.006,E2 -10896.006} C_VEL
LIN {X 0,Y 403.205,Z 460.255,A -85,B 0,C 180,E1 -10897.26,E2 -10897.26} C_VEL
LIN {X 0,Y 403.431,Z 453.953,A -85,B 0,C 180,E1 -10898.515,E2 -10898.515} C_VEL
LIN {X 0,Y 403.747,Z 447.794,A -85,B 0,C 180,E1 -10899.519,E2 -10899.519} C_VEL
LIN {X 0,Y 404.172,Z 441.335,A -85,B 0,C 180,E1 -10900.394,E2 -10900.394} C_VEL
LIN {X 0,Y 404.467,Z 434.741,A -85,B 0,C 180,E1 -10901.146,E2 -10901.146} C_VEL
LIN {X 0,Y 404.911,Z 426.776,A -85,B 0,C 180,E1 -10901.895,E2 -10901.895} C_VEL
LIN {X 0,Y 405.311,Z 418.581,A -85,B 0,C 180,E1 -10902.518,E2 -10902.518} C_VEL
LIN {X 0,Y 405.746,Z 410.338,A -85,B 0,C 180,E1 -10903.013,E2 -10903.013} C_VEL
LIN {X 0,Y 406.073,Z 400.695,A -85,B 0,C 180,E1 -10903.448,E2 -10903.448} C_VEL
LIN {X 0,Y 406.393,Z 391.624,A -85,B 0,C 180,E1 -10903.724,E2 -10903.724} C_VEL
LIN {X 0,Y 406.92,Z 339.825,A -85,B 0,C 180,E1 -10904.717,E2 -10904.717} C_VEL
LIN {X 0,Y 404.133,Z 314.746,A -85,B 0,C 180,E1 -10905.314,E2 -10905.314} C_VEL
LIN {X 0,Y 404.89,Z 298.987,A -85,B 0,C 180,E1 -10908.73,E2 -10908.73} C_VEL
LIN {X 0,Y 405.981,Z 281.06,A -85,B 0,C 180,E1 -10912.654,E2 -10912.654} C_VEL
LIN {X 0,Y 406.183,Z 276.37,A -85,B 0,C 180,E1 -10913.694,E2 -10913.694} C_VEL
LIN {X 0,Y 404.26,Z 264.942,A -85,B 0,C 180,E1 -10916.419,E2 -10916.419} C_VEL
LIN {X 0,Y 404.164,Z 264.955,A -85,B 0,C 180,E1 -10919.605,E2 -10919.605} C_VEL
LIN {X 0,Y 404.171,Z 264.954,A -85,B 0,C 180,E1 -10923.419,E2 -10923.419} C_VEL
LIN {X 0,Y 404.142,Z 264.952,A -85,B 0,C 180,E1 -10926.246,E2 -10926.246} C_VEL
LIN {X 0,Y 404.157,Z 264.95,A -85,B 0,C 180,E1 -10928.756,E2 -10928.756} C_VEL
LIN {X 0,Y 404.123,Z 264.961,A -85,B 0,C 180,E1 -10931.599,E2 -10931.599} C_VEL
LIN {X 0,Y 404.145,Z 264.951,A -85,B 0,C 180,E1 -10934.521,E2 -10934.521} C_VEL
LIN {X 0,Y 404.135,Z 264.957,A -85,B 0,C 180,E1 -10937.295,E2 -10937.295} C_VEL
LIN {X 0,Y 404.168,Z 264.951,A -85,B 0,C 180,E1 -10939.955,E2 -10939.955} C_VEL
LIN {X 0,Y 404.134,Z 264.955,A -85,B 0,C 180,E1 -10943.124,E2 -10943.124} C_VEL
LIN {X 0,Y 404.143,Z 264.953,A -85,B 0,C 180,E1 -10946.187,E2 -10946.187} C_VEL
LIN {X 0,Y 404.143,Z 264.957,A -85,B 0,C 180,E1 -10949.714,E2 -10949.714} C_VEL
LIN {X 0,Y 404.192,Z 264.948,A -85,B 0,C 180,E1 -10953.122,E2 -10953.122} C_VEL
LIN {X 0,Y 404.175,Z 264.952,A -85,B 0,C 180,E1 -10955.334,E2 -10955.334} C_VEL
LIN {X 0,Y 404.135,Z 264.953,A -85,B 0,C 180,E1 -10958.58,E2 -10958.58} C_VEL
LIN {X 0,Y 404.206,Z 264.949,A -85,B 0,C 180,E1 -10961.761,E2 -10961.761} C_VEL
LIN {X 0,Y 404.201,Z 264.945,A -85,B 0,C 180,E1 -10964.881,E2 -10964.881} C_VEL
LIN {X 0,Y 404.251,Z 264.941,A -85,B 0,C 180,E1 -10967.958,E2 -10967.958} C_VEL
LIN {X 0,Y 404.4,Z 264.921,A -85,B 0,C 180,E1 -10972.128,E2 -10972.128} C_VEL
LIN {X 0,Y 404.418,Z 264.92,A -85,B 0,C 180,E1 -10974.014,E2 -10974.014} C_VEL
LIN {X 0,Y 404.477,Z 264.913,A -85,B 0,C 180,E1 -10978.008,E2 -10978.008} C_VEL
LIN {X 0,Y 404.605,Z 264.897,A -85,B 0,C 180,E1 -10979.999,E2 -10979.999} C_VEL
LIN {X 0,Y 404.417,Z 264.919,A -85,B 0,C 180,E1 -10982.988,E2 -10982.988} C_VEL
LIN {X 0,Y 404.405,Z 264.92,A -85,B 0,C 180,E1 -10986.986,E2 -10986.986} C_VEL
LIN {X 0,Y 404.264,Z 264.94,A -85,B 0,C 180,E1 -10990.011,E2 -10990.011} C_VEL
LIN {X 0,Y 404.26,Z 264.94,A -85,B 0,C 180,E1 -10993.211,E2 -10993.211} C_VEL
LIN {X 0,Y 404.208,Z 264.945,A -85,B 0,C 180,E1 -10997.006,E2 -10997.006} C_VEL
LIN {X 0,Y 404.19,Z 264.947,A -85,B 0,C 180,E1 -11000.349,E2 -11000.349} C_VEL
LIN {X 0,Y 404.161,Z 264.956,A -85,B 0,C 180,E1 -11003.574,E2 -11003.574} C_VEL
LIN {X 0,Y 404.176,Z 264.953,A -85,B 0,C 180,E1 -11005.766,E2 -11005.766} C_VEL
LIN {X 0,Y 404.187,Z 264.949,A -85,B 0,C 180,E1 -11007.999,E2 -11007.999} C_VEL
LIN {X 0,Y 404.131,Z 264.959,A -85,B 0,C 180,E1 -11011.557,E2 -11011.557} C_VEL
LIN {X 0,Y 404.177,Z 264.949,A -85,B 0,C 180,E1 -11015.015,E2 -11015.015} C_VEL
LIN {X 0,Y 404.155,Z 264.951,A -85,B 0,C 180,E1 -11018.755,E2 -11018.755} C_VEL
LIN {X 0,Y 404.142,Z 264.958,A -85,B 0,C 180,E1 -11021.604,E2 -11021.604} C_VEL
LIN {X 0,Y 404.148,Z 264.952,A -85,B 0,C 180,E1 -11024.523,E2 -11024.523} C_VEL
LIN {X 0,Y 404.198,Z 264.948,A -85,B 0,C 180,E1 -11027.304,E2 -11027.304} C_VEL
LIN {X 0,Y 404.16,Z 264.954,A -85,B 0,C 180,E1 -11029.955,E2 -11029.955} C_VEL
LIN {X 0,Y 404.131,Z 264.955,A -85,B 0,C 180,E1 -11033.124,E2 -11033.124} C_VEL
LIN {X 0,Y 404.136,Z 264.955,A -85,B 0,C 180,E1 -11036.187,E2 -11036.187} C_VEL
LIN {X 0,Y 404.136,Z 264.959,A -85,B 0,C 180,E1 -11039.715,E2 -11039.715} C_VEL
LIN {X 0,Y 404.186,Z 264.948,A -85,B 0,C 180,E1 -11043.123,E2 -11043.123} C_VEL
LIN {X 0,Y 404.169,Z 264.952,A -85,B 0,C 180,E1 -11045.334,E2 -11045.334} C_VEL
LIN {X 0,Y 404.131,Z 264.954,A -85,B 0,C 180,E1 -11048.58,E2 -11048.58} C_VEL
LIN {X 0,Y 404.201,Z 264.951,A -85,B 0,C 180,E1 -11051.762,E2 -11051.762} C_VEL
LIN {X 0,Y 404.197,Z 264.946,A -85,B 0,C 180,E1 -11054.882,E2 -11054.882} C_VEL
LIN {X 0,Y 404.248,Z 264.943,A -85,B 0,C 180,E1 -11057.958,E2 -11057.958} C_VEL
LIN {X 0,Y 404.424,Z 264.92,A -85,B 0,C 180,E1 -11062.1,E2 -11062.1} C_VEL
LIN {X 0,Y 404.411,Z 264.922,A -85,B 0,C 180,E1 -11064.015,E2 -11064.015} C_VEL
LIN {X 0,Y 404.47,Z 264.915,A -85,B 0,C 180,E1 -11068.008,E2 -11068.008} C_VEL
LIN {X 0,Y 404.601,Z 264.899,A -85,B 0,C 180,E1 -11070,E2 -11070} C_VEL
LIN {X 0,Y 404.406,Z 264.92,A -85,B 0,C 180,E1 -11072.988,E2 -11072.988} C_VEL
LIN {X 0,Y 404.391,Z 264.922,A -85,B 0,C 180,E1 -11076.987,E2 -11076.987} C_VEL
LIN {X 0,Y 404.26,Z 264.941,A -85,B 0,C 180,E1 -11080.011,E2 -11080.011} C_VEL
LIN {X 0,Y 404.257,Z 264.94,A -85,B 0,C 180,E1 -11083.211,E2 -11083.211} C_VEL
LIN {X 0,Y 404.206,Z 264.945,A -85,B 0,C 180,E1 -11087.007,E2 -11087.007} C_VEL
LIN {X 0,Y 404.153,Z 264.953,A -85,B 0,C 180,E1 -11090.351,E2 -11090.351} C_VEL
LIN {X 0,Y 404.125,Z 264.955,A -85,B 0,C 180,E1 -11091.925,E2 -11091.925} C_VEL
LIN {X 0,Y 403.483,Z 265.035,A -85,B 0,C 180,E1 -11092.756,E2 -11092.756} C_VEL
LIN {X 0,Y 400.649,Z 265.392,A -85,B 0,C 180,E1 -11094.108,E2 -11094.108} C_VEL
LIN {X 0,Y 398.238,Z 265.694,A -85,B 0,C 180,E1 -11095.2,E2 -11095.2} C_VEL
LIN {X 0,Y 397.204,Z 265.821,A -85,B 0,C 180,E1 -11096.044,E2 -11096.044} C_VEL
LIN {X 0,Y 397.121,Z 265.829,A -85,B 0,C 180,E1 -11096.33,E2 -11096.33} C_VEL
LIN {X 0,Y 397.11,Z 265.83,A -85,B 0,C 180,E1 -11098.544,E2 -11098.544} C_VEL
LIN {X 0,Y 397.165,Z 265.971,A -85,B 0,C 180,E1 -11101.858,E2 -11101.858} C_VEL
LIN {X 0,Y 397.556,Z 270.91,A -85,B 0,C 180,E1 -11103.23,E2 -11103.23} C_VEL
LIN {X 0,Y 397.512,Z 272.152,A -85,B 0,C 180,E1 -11103.562,E2 -11103.562} C_VEL
LIN {X 0,Y 400.396,Z 288.321,A -85,B 0,C 180,E1 -11103.985,E2 -11103.985} C_VEL
LIN {X 0,Y 399.629,Z 348.588,A -85,B 0,C 180,E1 -11105.165,E2 -11105.165} C_VEL
LIN {X 0,Y 399.389,Z 358.576,A -85,B 0,C 180,E1 -11105.498,E2 -11105.498} C_VEL
LIN {X 0,Y 399.131,Z 370.636,A -85,B 0,C 180,E1 -11106.115,E2 -11106.115} C_VEL
LIN {X 0,Y 398.679,Z 380.461,A -85,B 0,C 180,E1 -11106.823,E2 -11106.823} C_VEL
LIN {X 0,Y 398.346,Z 388.462,A -85,B 0,C 180,E1 -11107.551,E2 -11107.551} C_VEL
LIN {X 0,Y 397.921,Z 395.839,A -85,B 0,C 180,E1 -11108.367,E2 -11108.367} C_VEL
LIN {X 0,Y 397.435,Z 403.36,A -85,B 0,C 180,E1 -11109.381,E2 -11109.381} C_VEL
LIN {X 0,Y 397.074,Z 409.793,A -85,B 0,C 180,E1 -11110.443,E2 -11110.443} C_VEL
LIN {X 0,Y 396.688,Z 415.839,A -85,B 0,C 180,E1 -11111.664,E2 -11111.664} C_VEL
LIN {X 0,Y 396.473,Z 420.512,A -85,B 0,C 180,E1 -11112.845,E2 -11112.845} C_VEL
LIN {X 0,Y 396.228,Z 424.924,A -85,B 0,C 180,E1 -11114.282,E2 -11114.282} C_VEL
LIN {X 0,Y 396.069,Z 427.092,A -85,B 0,C 180,E1 -11115.215,E2 -11115.215} C_VEL
LIN {X 0,Y 395.856,Z 429.65,A -85,B 0,C 180,E1 -11116.71,E2 -11116.71} C_VEL
LIN {X 0,Y 395.77,Z 431.008,A -85,B 0,C 180,E1 -11118.228,E2 -11118.228} C_VEL
LIN {X 0,Y 395.809,Z 431.233,A -85,B 0,C 180,E1 -11119.773,E2 -11119.773} C_VEL
LIN {X 0,Y 395.944,Z 430.067,A -85,B 0,C 180,E1 -11121.594,E2 -11121.594} C_VEL
LIN {X 0,Y 396.166,Z 428.083,A -85,B 0,C 180,E1 -11122.966,E2 -11122.966} C_VEL
LIN {X 0,Y 396.48,Z 424.269,A -85,B 0,C 180,E1 -11124.624,E2 -11124.624} C_VEL
LIN {X 0,Y 396.815,Z 420.077,A -85,B 0,C 180,E1 -11125.938,E2 -11125.938} C_VEL
LIN {X 0,Y 397.143,Z 415.695,A -85,B 0,C 180,E1 -11127.034,E2 -11127.034} C_VEL
LIN {X 0,Y 397.482,Z 410.67,A -85,B 0,C 180,E1 -11128.068,E2 -11128.068} C_VEL
LIN {X 0,Y 397.977,Z 403.946,A -85,B 0,C 180,E1 -11129.196,E2 -11129.196} C_VEL
LIN {X 0,Y 398.54,Z 396.56,A -85,B 0,C 180,E1 -11130.204,E2 -11130.204} C_VEL
LIN {X 0,Y 399.091,Z 388.557,A -85,B 0,C 180,E1 -11131.094,E2 -11131.094} C_VEL
LIN {X 0,Y 399.609,Z 378.201,A -85,B 0,C 180,E1 -11132.009,E2 -11132.009} C_VEL
LIN {X 0,Y 400.046,Z 367.784,A -85,B 0,C 180,E1 -11132.681,E2 -11132.681} C_VEL
LIN {X 0,Y 400.333,Z 358.015,A -85,B 0,C 180,E1 -11133.145,E2 -11133.145} C_VEL
LIN {X 0,Y 400.521,Z 349.021,A -85,B 0,C 180,E1 -11133.437,E2 -11133.437} C_VEL
LIN {X 0,Y 401.353,Z 287.51,A -85,B 0,C 180,E1 -11134.671,E2 -11134.671} C_VEL
LIN {X 0,Y 398.171,Z 272.383,A -85,B 0,C 180,E1 -11135.147,E2 -11135.147} C_VEL
LIN {X 0,Y 397.122,Z 265.833,A -85,B 0,C 180,E1 -11136.771,E2 -11136.771} C_VEL
LIN {X 0,Y 397.137,Z 265.836,A -85,B 0,C 180,E1 -11140.353,E2 -11140.353} C_VEL
LIN {X 0,Y 397.156,Z 265.826,A -85,B 0,C 180,E1 -11143.554,E2 -11143.554} C_VEL
LIN {X 0,Y 397.218,Z 265.821,A -85,B 0,C 180,E1 -11146.703,E2 -11146.703} C_VEL
LIN {X 0,Y 397.209,Z 265.819,A -85,B 0,C 180,E1 -11149.81,E2 -11149.81} C_VEL
LIN {X 0,Y 397.344,Z 265.804,A -85,B 0,C 180,E1 -11152.889,E2 -11152.889} C_VEL
LIN {X 0,Y 397.251,Z 265.812,A -85,B 0,C 180,E1 -11154.926,E2 -11154.926} C_VEL
LIN {X 0,Y 397.443,Z 265.786,A -85,B 0,C 180,E1 -11157.974,E2 -11157.974} C_VEL
LIN {X 0,Y 397.571,Z 265.774,A -85,B 0,C 180,E1 -11160.001,E2 -11160.001} C_VEL
LIN {X 0,Y 397.374,Z 265.797,A -85,B 0,C 180,E1 -11163.042,E2 -11163.042} C_VEL
LIN {X 0,Y 397.356,Z 265.798,A -85,B 0,C 180,E1 -11167.113,E2 -11167.113} C_VEL
LIN {X 0,Y 397.21,Z 265.819,A -85,B 0,C 180,E1 -11170.192,E2 -11170.192} C_VEL
LIN {X 0,Y 397.219,Z 265.814,A -85,B 0,C 180,E1 -11173.322,E2 -11173.322} C_VEL
LIN {X 0,Y 397.175,Z 265.818,A -85,B 0,C 180,E1 -11177.156,E2 -11177.156} C_VEL
LIN {X 0,Y 397.096,Z 265.827,A -85,B 0,C 180,E1 -11180.731,E2 -11180.731} C_VEL
LIN {X 0,Y 397.127,Z 265.828,A -85,B 0,C 180,E1 -11184.019,E2 -11184.019} C_VEL
LIN {X 0,Y 397.189,Z 265.819,A -85,B 0,C 180,E1 -11187.391,E2 -11187.391} C_VEL
LIN {X 0,Y 397.08,Z 265.836,A -85,B 0,C 180,E1 -11190.883,E2 -11190.883} C_VEL
LIN {X 0,Y 397.121,Z 265.829,A -85,B 0,C 180,E1 -11194.494,E2 -11194.494} C_VEL
LIN {X 0,Y 397.106,Z 265.83,A -85,B 0,C 180,E1 -11198.275,E2 -11198.275} C_VEL
LIN {X 0,Y 397.109,Z 265.83,A -85,B 0,C 180,E1 -11200.907,E2 -11200.907} C_VEL
LIN {X 0,Y 397.099,Z 265.829,A -85,B 0,C 180,E1 -11203.649,E2 -11203.649} C_VEL
LIN {X 0,Y 397.099,Z 265.833,A -85,B 0,C 180,E1 -11206.522,E2 -11206.522} C_VEL
LIN {X 0,Y 397.113,Z 265.836,A -85,B 0,C 180,E1 -11210.424,E2 -11210.424} C_VEL
LIN {X 0,Y 397.108,Z 265.835,A -85,B 0,C 180,E1 -11214.266,E2 -11214.266} C_VEL
LIN {X 0,Y 397.113,Z 265.833,A -85,B 0,C 180,E1 -11216.728,E2 -11216.728} C_VEL
LIN {X 0,Y 397.124,Z 265.834,A -85,B 0,C 180,E1 -11220.297,E2 -11220.297} C_VEL
LIN {X 0,Y 397.206,Z 265.952,A -85,B 0,C 180,E1 -11223.712,E2 -11223.712} C_VEL
LIN {X 0,Y 399.059,Z 276.23,A -85,B 0,C 180,E1 -11226.106,E2 -11226.106} C_VEL
LIN {X 0,Y 398.688,Z 285.042,A -85,B 0,C 180,E1 -11228.002,E2 -11228.002} C_VEL
LIN {X 0,Y 397.759,Z 302.525,A -85,B 0,C 180,E1 -11231.723,E2 -11231.723} C_VEL
LIN {X 0,Y 397.291,Z 312.665,A -85,B 0,C 180,E1 -11233.86,E2 -11233.86} C_VEL
LIN {X 0,Y 400.167,Z 333.886,A -85,B 0,C 180,E1 -11234.434,E2 -11234.434} C_VEL
LIN {X 0,Y 400.905,Z 343.329,A -85,B 0,C 180,E1 -11234.658,E2 -11234.658} C_VEL
LIN {X 0,Y 400.226,Z 391.087,A -85,B 0,C 180,E1 -11235.608,E2 -11235.608} C_VEL
LIN {X 0,Y 399.867,Z 400.616,A -85,B 0,C 180,E1 -11235.918,E2 -11235.918} C_VEL
LIN {X 0,Y 399.302,Z 411.688,A -85,B 0,C 180,E1 -11236.45,E2 -11236.45} C_VEL
LIN {X 0,Y 398.65,Z 421.87,A -85,B 0,C 180,E1 -11237.14,E2 -11237.14} C_VEL
LIN {X 0,Y 398.085,Z 430.493,A -85,B 0,C 180,E1 -11237.899,E2 -11237.899} C_VEL
LIN {X 0,Y 397.522,Z 438.638,A -85,B 0,C 180,E1 -11238.786,E2 -11238.786} C_VEL
LIN {X 0,Y 397.138,Z 444.521,A -85,B 0,C 180,E1 -11239.55,E2 -11239.55} C_VEL
LIN {X 0,Y 396.684,Z 451.086,A -85,B 0,C 180,E1 -11240.568,E2 -11240.568} C_VEL
LIN {X 0,Y 396.349,Z 456.558,A -85,B 0,C 180,E1 -11241.589,E2 -11241.589} C_VEL
LIN {X 0,Y 396.106,Z 462.121,A -85,B 0,C 180,E1 -11242.866,E2 -11242.866} C_VEL
LIN {X 0,Y 395.91,Z 465.743,A -85,B 0,C 180,E1 -11243.886,E2 -11243.886} C_VEL
LIN {X 0,Y 395.887,Z 469.925,A -85,B 0,C 180,E1 -11245.418,E2 -11245.418} C_VEL
LIN {X 0,Y 395.829,Z 472.823,A -85,B 0,C 180,E1 -11246.947,E2 -11246.947} C_VEL
LIN {X 0,Y 395.9,Z 474.02,A -85,B 0,C 180,E1 -11247.966,E2 -11247.966} C_VEL
LIN {X 0,Y 395.855,Z 474.721,A -85,B 0,C 180,E1 -11248.983,E2 -11248.983} C_VEL
LIN {X 0,Y 395.87,Z 474.945,A -85,B 0,C 180,E1 -11250,E2 -11250} C_VEL
LIN {X 0,Y 395.863,Z 474.64,A -85,B 0,C 180,E1 -11251.017,E2 -11251.017} C_VEL
LIN {X 0,Y 395.905,Z 473.736,A -85,B 0,C 180,E1 -11252.035,E2 -11252.035} C_VEL
LIN {X 0,Y 395.866,Z 472.316,A -85,B 0,C 180,E1 -11253.053,E2 -11253.053} C_VEL
LIN {X 0,Y 395.893,Z 469.207,A -85,B 0,C 180,E1 -11254.582,E2 -11254.582} C_VEL
LIN {X 0,Y 395.946,Z 464.097,A -85,B 0,C 180,E1 -11256.28,E2 -11256.28} C_VEL
LIN {X 0,Y 396.133,Z 459.704,A -85,B 0,C 180,E1 -11257.39,E2 -11257.39} C_VEL
LIN {X 0,Y 396.394,Z 453.367,A -85,B 0,C 180,E1 -11258.668,E2 -11258.668} C_VEL
LIN {X 0,Y 396.725,Z 447.166,A -85,B 0,C 180,E1 -11259.689,E2 -11259.689} C_VEL
LIN {X 0,Y 397.163,Z 440.657,A -85,B 0,C 180,E1 -11260.579,E2 -11260.579} C_VEL
LIN {X 0,Y 397.508,Z 434.006,A -85,B 0,C 180,E1 -11261.344,E2 -11261.344} C_VEL
LIN {X 0,Y 397.938,Z 425.961,A -85,B 0,C 180,E1 -11262.106,E2 -11262.106} C_VEL
LIN {X 0,Y 398.378,Z 417.665,A -85,B 0,C 180,E1 -11262.74,E2 -11262.74} C_VEL
LIN {X 0,Y 398.762,Z 409.262,A -85,B 0,C 180,E1 -11263.245,E2 -11263.245} C_VEL
LIN {X 0,Y 399.167,Z 399.39,A -85,B 0,C 180,E1 -11263.685,E2 -11263.685} C_VEL
LIN {X 0,Y 399.514,Z 388.596,A -85,B 0,C 180,E1 -11263.998,E2 -11263.998} C_VEL
LIN {X 0,Y 399.947,Z 339.525,A -85,B 0,C 180,E1 -11264.945,E2 -11264.945} C_VEL
LIN {X 0,Y 397.142,Z 314.366,A -85,B 0,C 180,E1 -11265.558,E2 -11265.558} C_VEL
LIN {X 0,Y 397.885,Z 298.457,A -85,B 0,C 180,E1 -11269.073,E2 -11269.073} C_VEL
LIN {X 0,Y 398.875,Z 282.943,A -85,B 0,C 180,E1 -11272.533,E2 -11272.533} C_VEL
LIN {X 0,Y 399.132,Z 276.94,A -85,B 0,C 180,E1 -11273.89,E2 -11273.89} C_VEL
LIN {X 0,Y 397.204,Z 265.82,A -85,B 0,C 180,E1 -11276.607,E2 -11276.607} C_VEL
LIN {X 0,Y 397.106,Z 265.831,A -85,B 0,C 180,E1 -11279.864,E2 -11279.864} C_VEL
LIN {X 0,Y 397.119,Z 265.831,A -85,B 0,C 180,E1 -11283.717,E2 -11283.717} C_VEL
LIN {X 0,Y 397.094,Z 265.833,A -85,B 0,C 180,E1 -11287.208,E2 -11287.208} C_VEL
LIN {X 0,Y 397.102,Z 265.829,A -85,B 0,C 180,E1 -11290.445,E2 -11290.445} C_VEL
LIN {X 0,Y 397.101,Z 265.835,A -85,B 0,C 180,E1 -11293.648,E2 -11293.648} C_VEL
LIN {X 0,Y 397.101,Z 265.829,A -85,B 0,C 180,E1 -11296.52,E2 -11296.52} C_VEL
LIN {X 0,Y 397.111,Z 265.828,A -85,B 0,C 180,E1 -11300.422,E2 -11300.422} C_VEL
LIN {X 0,Y 397.106,Z 265.829,A -85,B 0,C 180,E1 -11304.265,E2 -11304.265} C_VEL
LIN {X 0,Y 397.112,Z 265.828,A -85,B 0,C 180,E1 -11306.726,E2 -11306.726} C_VEL
LIN {X 0,Y 397.122,Z 265.827,A -85,B 0,C 180,E1 -11310.295,E2 -11310.295} C_VEL
LIN {X 0,Y 397.192,Z 265.818,A -85,B 0,C 180,E1 -11312.609,E2 -11312.609} C_VEL
LIN {X 0,Y 397.13,Z 265.828,A -85,B 0,C 180,E1 -11315.981,E2 -11315.981} C_VEL
LIN {X 0,Y 397.135,Z 265.83,A -85,B 0,C 180,E1 -11319.704,E2 -11319.704} C_VEL
LIN {X 0,Y 397.178,Z 265.82,A -85,B 0,C 180,E1 -11322.844,E2 -11322.844} C_VEL
LIN {X 0,Y 397.225,Z 265.814,A -85,B 0,C 180,E1 -11326.702,E2 -11326.702} C_VEL
LIN {X 0,Y 397.213,Z 265.819,A -85,B 0,C 180,E1 -11329.808,E2 -11329.808} C_VEL
LIN {X 0,Y 397.347,Z 265.799,A -85,B 0,C 180,E1 -11332.887,E2 -11332.887} C_VEL
LIN {X 0,Y 397.25,Z 265.811,A -85,B 0,C 180,E1 -11334.924,E2 -11334.924} C_VEL
LIN {X 0,Y 397.446,Z 265.789,A -85,B 0,C 180,E1 -11337.972,E2 -11337.972} C_VEL
LIN {X 0,Y 397.575,Z 265.773,A -85,B 0,C 180,E1 -11339.999,E2 -11339.999} C_VEL
LIN {X 0,Y 397.376,Z 265.796,A -85,B 0,C 180,E1 -11343.041,E2 -11343.041} C_VEL
LIN {X 0,Y 397.357,Z 265.799,A -85,B 0,C 180,E1 -11347.111,E2 -11347.111} C_VEL
LIN {X 0,Y 397.221,Z 265.816,A -85,B 0,C 180,E1 -11350.19,E2 -11350.19} C_VEL
LIN {X 0,Y 397.22,Z 265.818,A -85,B 0,C 180,E1 -11353.32,E2 -11353.32} C_VEL
LIN {X 0,Y 397.175,Z 265.822,A -85,B 0,C 180,E1 -11357.154,E2 -11357.154} C_VEL
LIN {X 0,Y 397.119,Z 265.827,A -85,B 0,C 180,E1 -11360.728,E2 -11360.728} C_VEL
LIN {X 0,Y 397.125,Z 265.829,A -85,B 0,C 180,E1 -11364.018,E2 -11364.018} C_VEL
LIN {X 0,Y 397.186,Z 265.822,A -85,B 0,C 180,E1 -11367.389,E2 -11367.389} C_VEL
LIN {X 0,Y 397.07,Z 265.834,A -85,B 0,C 180,E1 -11370.882,E2 -11370.882} C_VEL
LIN {X 0,Y 397.117,Z 265.828,A -85,B 0,C 180,E1 -11374.493,E2 -11374.493} C_VEL
LIN {X 0,Y 397.101,Z 265.831,A -85,B 0,C 180,E1 -11378.274,E2 -11378.274} C_VEL
LIN {X 0,Y 397.104,Z 265.829,A -85,B 0,C 180,E1 -11380.905,E2 -11380.905} C_VEL
LIN {X 0,Y 397.098,Z 265.836,A -85,B 0,C 180,E1 -11383.647,E2 -11383.647} C_VEL
LIN {X 0,Y 397.151,Z 265.824,A -85,B 0,C 180,E1 -11386.512,E2 -11386.512} C_VEL
LIN {X 0,Y 397.114,Z 265.833,A -85,B 0,C 180,E1 -11389.55,E2 -11389.55} C_VEL
LIN {X 0,Y 397.089,Z 265.831,A -85,B 0,C 180,E1 -11392.79,E2 -11392.79} C_VEL
LIN {X 0,Y 397.11,Z 265.83,A -85,B 0,C 180,E1 -11396.282,E2 -11396.282} C_VEL
LIN {X 0,Y 397.096,Z 265.832,A -85,B 0,C 180,E1 -11400.135,E2 -11400.135} C_VEL
LIN {X 0,Y 397.185,Z 265.819,A -85,B 0,C 180,E1 -11402.61,E2 -11402.61} C_VEL
LIN {X 0,Y 397.125,Z 265.83,A -85,B 0,C 180,E1 -11405.981,E2 -11405.981} C_VEL
LIN {X 0,Y 397.136,Z 265.832,A -85,B 0,C 180,E1 -11409.702,E2 -11409.702} C_VEL
LIN {X 0,Y 397.173,Z 265.821,A -85,B 0,C 180,E1 -11412.845,E2 -11412.845} C_VEL
LIN {X 0,Y 397.22,Z 265.815,A -85,B 0,C 180,E1 -11416.702,E2 -11416.702} C_VEL
LIN {X 0,Y 397.21,Z 265.821,A -85,B 0,C 180,E1 -11419.809,E2 -11419.809} C_VEL
LIN {X 0,Y 397.353,Z 265.798,A -85,B 0,C 180,E1 -11422.888,E2 -11422.888} C_VEL
LIN {X 0,Y 397.243,Z 265.812,A -85,B 0,C 180,E1 -11424.925,E2 -11424.925} C_VEL
LIN {X 0,Y 397.439,Z 265.791,A -85,B 0,C 180,E1 -11427.973,E2 -11427.973} C_VEL
LIN {X 0,Y 397.571,Z 265.775,A -85,B 0,C 180,E1 -11430,E2 -11430} C_VEL
LIN {X 0,Y 397.366,Z 265.797,A -85,B 0,C 180,E1 -11433.041,E2 -11433.041} C_VEL
LIN {X 0,Y 397.36,Z 265.8,A -85,B 0,C 180,E1 -11436.091,E2 -11436.091} C_VEL
LIN {X 0,Y 397.248,Z 265.812,A -85,B 0,C 180,E1 -11439.161,E2 -11439.161} C_VEL
LIN {X 0,Y 397.219,Z 265.817,A -85,B 0,C 180,E1 -11442.258,E2 -11442.258} C_VEL
LIN {X 0,Y 397.17,Z 265.824,A -85,B 0,C 180,E1 -11445.392,E2 -11445.392} C_VEL
LIN {X 0,Y 397.151,Z 265.824,A -85,B 0,C 180,E1 -11448.573,E2 -11448.573} C_VEL
LIN {X 0,Y 397.081,Z 265.836,A -85,B 0,C 180,E1 -11451.918,E2 -11451.918} C_VEL
LIN {X 0,Y 397.14,Z 265.828,A -85,B 0,C 180,E1 -11455.512,E2 -11455.512} C_VEL
LIN {X 0,Y 397.121,Z 265.829,A -85,B 0,C 180,E1 -11456.33,E2 -11456.33} C_VEL
LIN {X 0,Y 396.448,Z 265.913,A -85,B 0,C 180,E1 -11457.177,E2 -11457.177} C_VEL
LIN {X 0,Y 393.562,Z 266.272,A -85,B 0,C 180,E1 -11458.552,E2 -11458.552} C_VEL
LIN {X 0,Y 391.131,Z 266.578,A -85,B 0,C 180,E1 -11459.664,E2 -11459.664} C_VEL
LIN {X 0,Y 390.106,Z 266.702,A -85,B 0,C 180,E1 -11460.524,E2 -11460.524} C_VEL
LIN {X 0,Y 390.033,Z 266.711,A -85,B 0,C 180,E1 -11460.815,E2 -11460.815} C_VEL
LIN {X 0,Y 390.112,Z 266.823,A -85,B 0,C 180,E1 -11461.725,E2 -11461.725} C_VEL
LIN {X 0,Y 390.562,Z 271.247,A -85,B 0,C 180,E1 -11462.978,E2 -11462.978} C_VEL
LIN {X 0,Y 390.558,Z 272.74,A -85,B 0,C 180,E1 -11463.325,E2 -11463.325} C_VEL
LIN {X 0,Y 393.501,Z 289.142,A -85,B 0,C 180,E1 -11463.766,E2 -11463.766} C_VEL
LIN {X 0,Y 392.689,Z 349.569,A -85,B 0,C 180,E1 -11464.977,E2 -11464.977} C_VEL
LIN {X 0,Y 392.419,Z 360.379,A -85,B 0,C 180,E1 -11465.358,E2 -11465.358} C_VEL
LIN {X 0,Y 392.06,Z 372.502,A -85,B 0,C 180,E1 -11466.03,E2 -11466.03} C_VEL
LIN {X 0,Y 391.657,Z 381.543,A -85,B 0,C 180,E1 -11466.709,E2 -11466.709} C_VEL
LIN {X 0,Y 391.324,Z 389.62,A -85,B 0,C 180,E1 -11467.471,E2 -11467.471} C_VEL
LIN {X 0,Y 390.857,Z 397.368,A -85,B 0,C 180,E1 -11468.364,E2 -11468.364} C_VEL
LIN {X 0,Y 390.312,Z 405.467,A -85,B 0,C 180,E1 -11469.511,E2 -11469.511} C_VEL
LIN {X 0,Y 389.87,Z 413.605,A -85,B 0,C 180,E1 -11471.007,E2 -11471.007} C_VEL
LIN {X 0,Y 389.472,Z 419.052,A -85,B 0,C 180,E1 -11472.284,E2 -11472.284} C_VEL
LIN {X 0,Y 389.203,Z 423.951,A -85,B 0,C 180,E1 -11473.757,E2 -11473.757} C_VEL
LIN {X 0,Y 388.979,Z 427.516,A -85,B 0,C 180,E1 -11475.201,E2 -11475.201} C_VEL
LIN {X 0,Y 388.781,Z 429.919,A -85,B 0,C 180,E1 -11476.614,E2 -11476.614} C_VEL
LIN {X 0,Y 388.684,Z 431.301,A -85,B 0,C 180,E1 -11478.011,E2 -11478.011} C_VEL
LIN {X 0,Y 388.717,Z 431.742,A -85,B 0,C 180,E1 -11479.406,E2 -11479.406} C_VEL
LIN {X 0,Y 388.784,Z 431.066,A -85,B 0,C 180,E1 -11481.013,E2 -11481.013} C_VEL
LIN {X 0,Y 389.015,Z 429.146,A -85,B 0,C 180,E1 -11482.645,E2 -11482.645} C_VEL
LIN {X 0,Y 389.338,Z 425.848,A -85,B 0,C 180,E1 -11484.319,E2 -11484.319} C_VEL
LIN {X 0,Y 389.794,Z 420.719,A -85,B 0,C 180,E1 -11486.033,E2 -11486.033} C_VEL
LIN {X 0,Y 390.177,Z 415.74,A -85,B 0,C 180,E1 -11487.293,E2 -11487.293} C_VEL
LIN {X 0,Y 390.649,Z 409.5,A -85,B 0,C 180,E1 -11488.553,E2 -11488.553} C_VEL
LIN {X 0,Y 391.144,Z 403.173,A -85,B 0,C 180,E1 -11489.591,E2 -11489.591} C_VEL
LIN {X 0,Y 391.861,Z 394.53,A -85,B 0,C 180,E1 -11490.744,E2 -11490.744} C_VEL
LIN {X 0,Y 392.468,Z 385.123,A -85,B 0,C 180,E1 -11491.717,E2 -11491.717} C_VEL
LIN {X 0,Y 392.872,Z 376.601,A -85,B 0,C 180,E1 -11492.417,E2 -11492.417} C_VEL
LIN {X 0,Y 393.272,Z 367.908,A -85,B 0,C 180,E1 -11492.975,E2 -11492.975} C_VEL
LIN {X 0,Y 393.529,Z 358.419,A -85,B 0,C 180,E1 -11493.434,E2 -11493.434} C_VEL
LIN {X 0,Y 393.773,Z 348.684,A -85,B 0,C 180,E1 -11493.751,E2 -11493.751} C_VEL
LIN {X 0,Y 394.637,Z 288.474,A -85,B 0,C 180,E1 -11494.98,E2 -11494.98} C_VEL
LIN {X 0,Y 391.206,Z 272.816,A -85,B 0,C 180,E1 -11495.49,E2 -11495.49} C_VEL
LIN {X 0,Y 390.079,Z 266.711,A -85,B 0,C 180,E1 -11497.039,E2 -11497.039} C_VEL
LIN {X 0,Y 390.093,Z 266.712,A -85,B 0,C 180,E1 -11499.984,E2 -11499.984} C_VEL
LIN {X 0,Y 390.128,Z 266.702,A -85,B 0,C 180,E1 -11503.249,E2 -11503.249} C_VEL
LIN {X 0,Y 390.184,Z 266.697,A -85,B 0,C 180,E1 -11506.562,E2 -11506.562} C_VEL
LIN {X 0,Y 390.159,Z 266.697,A -85,B 0,C 180,E1 -11509.624,E2 -11509.624} C_VEL
LIN {X 0,Y 390.295,Z 266.682,A -85,B 0,C 180,E1 -11512.76,E2 -11512.76} C_VEL
LIN {X 0,Y 390.223,Z 266.688,A -85,B 0,C 180,E1 -11514.834,E2 -11514.834} C_VEL
LIN {X 0,Y 390.412,Z 266.662,A -85,B 0,C 180,E1 -11517.938,E2 -11517.938} C_VEL
LIN {X 0,Y 390.541,Z 266.65,A -85,B 0,C 180,E1 -11520.001,E2 -11520.001} C_VEL
LIN {X 0,Y 390.308,Z 266.677,A -85,B 0,C 180,E1 -11523.097,E2 -11523.097} C_VEL
LIN {X 0,Y 390.322,Z 266.677,A -85,B 0,C 180,E1 -11526.203,E2 -11526.203} C_VEL
LIN {X 0,Y 390.307,Z 266.675,A -85,B 0,C 180,E1 -11528.283,E2 -11528.283} C_VEL
LIN {X 0,Y 390.163,Z 266.692,A -85,B 0,C 180,E1 -11532.484,E2 -11532.484} C_VEL
LIN {X 0,Y 390.132,Z 266.697,A -85,B 0,C 180,E1 -11535.678,E2 -11535.678} C_VEL
LIN {X 0,Y 390.099,Z 266.703,A -85,B 0,C 180,E1 -11538.923,E2 -11538.923} C_VEL
LIN {X 0,Y 390.033,Z 266.709,A -85,B 0,C 180,E1 -11542.235,E2 -11542.235} C_VEL
LIN {X 0,Y 390.113,Z 266.694,A -85,B 0,C 180,E1 -11545.744,E2 -11545.744} C_VEL
LIN {X 0,Y 390.06,Z 266.701,A -85,B 0,C 180,E1 -11549.11,E2 -11549.11} C_VEL
LIN {X 0,Y 390.039,Z 266.708,A -85,B 0,C 180,E1 -11552.723,E2 -11552.723} C_VEL
LIN {X 0,Y 390.053,Z 266.709,A -85,B 0,C 180,E1 -11555.827,E2 -11555.827} C_VEL
LIN {X 0,Y 390.07,Z 266.707,A -85,B 0,C 180,E1 -11559.22,E2 -11559.22} C_VEL
LIN {X 0,Y 390.077,Z 266.711,A -85,B 0,C 180,E1 -11562.381,E2 -11562.381} C_VEL
LIN {X 0,Y 390.052,Z 266.712,A -85,B 0,C 180,E1 -11566.115,E2 -11566.115} C_VEL
LIN {X 0,Y 390.055,Z 266.709,A -85,B 0,C 180,E1 -11569.562,E2 -11569.562} C_VEL
LIN {X 0,Y 390.044,Z 266.717,A -85,B 0,C 180,E1 -11572.45,E2 -11572.45} C_VEL
LIN {X 0,Y 390.067,Z 266.71,A -85,B 0,C 180,E1 -11576.046,E2 -11576.046} C_VEL
LIN {X 0,Y 390.046,Z 266.714,A -85,B 0,C 180,E1 -11579.87,E2 -11579.87} C_VEL
LIN {X 0,Y 390.122,Z 266.703,A -85,B 0,C 180,E1 -11583.416,E2 -11583.416} C_VEL
LIN {X 0,Y 391.902,Z 276.04,A -85,B 0,C 180,E1 -11585.641,E2 -11585.641} C_VEL
LIN {X 0,Y 392.147,Z 279.472,A -85,B 0,C 180,E1 -11586.424,E2 -11586.424} C_VEL
LIN {X 0,Y 391.201,Z 294.891,A -85,B 0,C 180,E1 -11589.784,E2 -11589.784} C_VEL
LIN {X 0,Y 390.431,Z 309.293,A -85,B 0,C 180,E1 -11592.887,E2 -11592.887} C_VEL
LIN {X 0,Y 390.311,Z 312.193,A -85,B 0,C 180,E1 -11593.509,E2 -11593.509} C_VEL
LIN {X 0,Y 393.204,Z 332.556,A -85,B 0,C 180,E1 -11594.082,E2 -11594.082} C_VEL
LIN {X 0,Y 394.139,Z 343.507,A -85,B 0,C 180,E1 -11594.355,E2 -11594.355} C_VEL
LIN {X 0,Y 393.405,Z 391.156,A -85,B 0,C 180,E1 -11595.33,E2 -11595.33} C_VEL
LIN {X 0,Y 392.972,Z 401.854,A -85,B 0,C 180,E1 -11595.699,E2 -11595.699} C_VEL
LIN {X 0,Y 392.375,Z 412.853,A -85,B 0,C 180,E1 -11596.272,E2 -11596.272} C_VEL
LIN {X 0,Y 391.639,Z 423.342,A -85,B 0,C 180,E1 -11597.038,E2 -11597.038} C_VEL
LIN {X 0,Y 391.069,Z 431.634,A -85,B 0,C 180,E1 -11597.81,E2 -11597.81} C_VEL
LIN {X 0,Y 390.479,Z 439.525,A -85,B 0,C 180,E1 -11598.713,E2 -11598.713} C_VEL
LIN {X 0,Y 390.013,Z 446.067,A -85,B 0,C 180,E1 -11599.619,E2 -11599.619} C_VEL
LIN {X 0,Y 389.579,Z 452.315,A -85,B 0,C 180,E1 -11600.657,E2 -11600.657} C_VEL
LIN {X 0,Y 389.192,Z 458.717,A -85,B 0,C 180,E1 -11601.956,E2 -11601.956} C_VEL
LIN {X 0,Y 388.929,Z 463.809,A -85,B 0,C 180,E1 -11603.255,E2 -11603.255} C_VEL
LIN {X 0,Y 388.786,Z 468.401,A -85,B 0,C 180,E1 -11604.815,E2 -11604.815} C_VEL
LIN {X 0,Y 388.757,Z 470.762,A -85,B 0,C 180,E1 -11605.854,E2 -11605.854} C_VEL
LIN {X 0,Y 388.73,Z 472.482,A -85,B 0,C 180,E1 -11606.891,E2 -11606.891} C_VEL
LIN {X 0,Y 388.812,Z 473.655,A -85,B 0,C 180,E1 -11607.929,E2 -11607.929} C_VEL
LIN {X 0,Y 388.783,Z 474.336,A -85,B 0,C 180,E1 -11608.964,E2 -11608.964} C_VEL
LIN {X 0,Y 388.794,Z 474.538,A -85,B 0,C 180,E1 -11610,E2 -11610} C_VEL
LIN {X 0,Y 388.792,Z 474.226,A -85,B 0,C 180,E1 -11611.036,E2 -11611.036} C_VEL
LIN {X 0,Y 388.837,Z 473.308,A -85,B 0,C 180,E1 -11612.072,E2 -11612.072} C_VEL
LIN {X 0,Y 388.768,Z 471.863,A -85,B 0,C 180,E1 -11613.109,E2 -11613.109} C_VEL
LIN {X 0,Y 388.823,Z 468.731,A -85,B 0,C 180,E1 -11614.666,E2 -11614.666} C_VEL
LIN {X 0,Y 388.835,Z 464.187,A -85,B 0,C 180,E1 -11616.226,E2 -11616.226} C_VEL
LIN {X 0,Y 389.057,Z 459.126,A -85,B 0,C 180,E1 -11617.525,E2 -11617.525} C_VEL
LIN {X 0,Y 389.364,Z 452.748,A -85,B 0,C 180,E1 -11618.826,E2 -11618.826} C_VEL
LIN {X 0,Y 389.692,Z 446.493,A -85,B 0,C 180,E1 -11619.865,E2 -11619.865} C_VEL
LIN {X 0,Y 390.097,Z 439.918,A -85,B 0,C 180,E1 -11620.773,E2 -11620.773} C_VEL
LIN {X 0,Y 390.553,Z 431.953,A -85,B 0,C 180,E1 -11621.68,E2 -11621.68} C_VEL
LIN {X 0,Y 391.142,Z 422.041,A -85,B 0,C 180,E1 -11622.583,E2 -11622.583} C_VEL
LIN {X 0,Y 391.748,Z 410.443,A -85,B 0,C 180,E1 -11623.355,E2 -11623.355} C_VEL
LIN {X 0,Y 392.109,Z 401.124,A -85,B 0,C 180,E1 -11623.804,E2 -11623.804} C_VEL
LIN {X 0,Y 392.493,Z 391.469,A -85,B 0,C 180,E1 -11624.121,E2 -11624.121} C_VEL
LIN {X 0,Y 393.069,Z 340.405,A -85,B 0,C 180,E1 -11625.146,E2 -11625.146} C_VEL
LIN {X 0,Y 390.116,Z 313.973,A -85,B 0,C 180,E1 -11625.812,E2 -11625.812} C_VEL
LIN {X 0,Y 390.913,Z 297.929,A -85,B 0,C 180,E1 -11629.427,E2 -11629.427} C_VEL
LIN {X 0,Y 392.004,Z 282.401,A -85,B 0,C 180,E1 -11632.951,E2 -11632.951} C_VEL
LIN {X 0,Y 392.158,Z 278.129,A -85,B 0,C 180,E1 -11633.937,E2 -11633.937} C_VEL
LIN {X 0,Y 390.154,Z 266.699,A -85,B 0,C 180,E1 -11636.765,E2 -11636.765} C_VEL
LIN {X 0,Y 390.04,Z 266.709,A -85,B 0,C 180,E1 -11640.299,E2 -11640.299} C_VEL
LIN {X 0,Y 390.069,Z 266.707,A -85,B 0,C 180,E1 -11644.024,E2 -11644.024} C_VEL
LIN {X 0,Y 390.044,Z 266.715,A -85,B 0,C 180,E1 -11647.55,E2 -11647.55} C_VEL
LIN {X 0,Y 390.057,Z 266.707,A -85,B 0,C 180,E1 -11650.821,E2 -11650.821} C_VEL
LIN {X 0,Y 390.054,Z 266.71,A -85,B 0,C 180,E1 -11653.885,E2 -11653.885} C_VEL
LIN {X 0,Y 390.056,Z 266.707,A -85,B 0,C 180,E1 -11656.789,E2 -11656.789} C_VEL
LIN {X 0,Y 390.055,Z 266.714,A -85,B 0,C 180,E1 -11659.56,E2 -11659.56} C_VEL
LIN {X 0,Y 390.04,Z 266.709,A -85,B 0,C 180,E1 -11662.449,E2 -11662.449} C_VEL
LIN {X 0,Y 390.066,Z 266.708,A -85,B 0,C 180,E1 -11665.975,E2 -11665.975} C_VEL
LIN {X 0,Y 390.044,Z 266.712,A -85,B 0,C 180,E1 -11669.868,E2 -11669.868} C_VEL
LIN {X 0,Y 390.111,Z 266.703,A -85,B 0,C 180,E1 -11673.231,E2 -11673.231} C_VEL
LIN {X 0,Y 390.104,Z 266.701,A -85,B 0,C 180,E1 -11676.749,E2 -11676.749} C_VEL
LIN {X 0,Y 390.1,Z 266.704,A -85,B 0,C 180,E1 -11679.982,E2 -11679.982} C_VEL
LIN {X 0,Y 390.134,Z 266.7,A -85,B 0,C 180,E1 -11683.247,E2 -11683.247} C_VEL
LIN {X 0,Y 390.191,Z 266.69,A -85,B 0,C 180,E1 -11686.561,E2 -11686.561} C_VEL
LIN {X 0,Y 390.2,Z 266.689,A -85,B 0,C 180,E1 -11690.67,E2 -11690.67} C_VEL
LIN {X 0,Y 390.322,Z 266.678,A -85,B 0,C 180,E1 -11693.797,E2 -11693.797} C_VEL
LIN {X 0,Y 390.415,Z 266.665,A -85,B 0,C 180,E1 -11697.936,E2 -11697.936} C_VEL
LIN {X 0,Y 390.544,Z 266.649,A -85,B 0,C 180,E1 -11699.999,E2 -11699.999} C_VEL
LIN {X 0,Y 390.31,Z 266.677,A -85,B 0,C 180,E1 -11703.096,E2 -11703.096} C_VEL
LIN {X 0,Y 390.303,Z 266.676,A -85,B 0,C 180,E1 -11706.654,E2 -11706.654} C_VEL
LIN {X 0,Y 390.203,Z 266.692,A -85,B 0,C 180,E1 -11709.328,E2 -11709.328} C_VEL
LIN {X 0,Y 390.171,Z 266.693,A -85,B 0,C 180,E1 -11712.482,E2 -11712.482} C_VEL
LIN {X 0,Y 390.133,Z 266.704,A -85,B 0,C 180,E1 -11715.676,E2 -11715.676} C_VEL
LIN {X 0,Y 390.109,Z 266.701,A -85,B 0,C 180,E1 -11718.921,E2 -11718.921} C_VEL
LIN {X 0,Y 390.04,Z 266.71,A -85,B 0,C 180,E1 -11722.233,E2 -11722.233} C_VEL
LIN {X 0,Y 390.112,Z 266.705,A -85,B 0,C 180,E1 -11725.743,E2 -11725.743} C_VEL
LIN {X 0,Y 390.05,Z 266.709,A -85,B 0,C 180,E1 -11729.109,E2 -11729.109} C_VEL
LIN {X 0,Y 390.034,Z 266.71,A -85,B 0,C 180,E1 -11732.721,E2 -11732.721} C_VEL
LIN {X 0,Y 390.049,Z 266.712,A -85,B 0,C 180,E1 -11735.825,E2 -11735.825} C_VEL
LIN {X 0,Y 390.066,Z 266.708,A -85,B 0,C 180,E1 -11739.219,E2 -11739.219} C_VEL
LIN {X 0,Y 390.073,Z 266.706,A -85,B 0,C 180,E1 -11742.38,E2 -11742.38} C_VEL
LIN {X 0,Y 390.093,Z 266.705,A -85,B 0,C 180,E1 -11746.106,E2 -11746.106} C_VEL
LIN {X 0,Y 390.074,Z 266.706,A -85,B 0,C 180,E1 -11749.174,E2 -11749.174} C_VEL
LIN {X 0,Y 390.038,Z 266.71,A -85,B 0,C 180,E1 -11752.448,E2 -11752.448} C_VEL
LIN {X 0,Y 390.059,Z 266.71,A -85,B 0,C 180,E1 -11756.045,E2 -11756.045} C_VEL
LIN {X 0,Y 390.037,Z 266.714,A -85,B 0,C 180,E1 -11759.869,E2 -11759.869} C_VEL
LIN {X 0,Y 390.104,Z 266.703,A -85,B 0,C 180,E1 -11763.231,E2 -11763.231} C_VEL
LIN {X 0,Y 390.098,Z 266.702,A -85,B 0,C 180,E1 -11766.75,E2 -11766.75} C_VEL
LIN {X 0,Y 390.098,Z 266.705,A -85,B 0,C 180,E1 -11769.983,E2 -11769.983} C_VEL
LIN {X 0,Y 390.129,Z 266.7,A -85,B 0,C 180,E1 -11773.248,E2 -11773.248} C_VEL
LIN {X 0,Y 390.186,Z 266.692,A -85,B 0,C 180,E1 -11776.561,E2 -11776.561} C_VEL
LIN {X 0,Y 390.197,Z 266.69,A -85,B 0,C 180,E1 -11780.671,E2 -11780.671} C_VEL
LIN {X 0,Y 390.308,Z 266.676,A -85,B 0,C 180,E1 -11782.759,E2 -11782.759} C_VEL
LIN {X 0,Y 390.215,Z 266.688,A -85,B 0,C 180,E1 -11784.833,E2 -11784.833} C_VEL
LIN {X 0,Y 390.408,Z 266.667,A -85,B 0,C 180,E1 -11787.937,E2 -11787.937} C_VEL
LIN {X 0,Y 390.54,Z 266.65,A -85,B 0,C 180,E1 -11790,E2 -11790} C_VEL
LIN {X 0,Y 390.301,Z 266.678,A -85,B 0,C 180,E1 -11793.096,E2 -11793.096} C_VEL
LIN {X 0,Y 390.314,Z 266.677,A -85,B 0,C 180,E1 -11796.202,E2 -11796.202} C_VEL
LIN {X 0,Y 390.2,Z 266.691,A -85,B 0,C 180,E1 -11799.328,E2 -11799.328} C_VEL
LIN {X 0,Y 390.168,Z 266.694,A -85,B 0,C 180,E1 -11802.483,E2 -11802.483} C_VEL
LIN {X 0,Y 390.13,Z 266.704,A -85,B 0,C 180,E1 -11805.677,E2 -11805.677} C_VEL
LIN {X 0,Y 390.095,Z 266.703,A -85,B 0,C 180,E1 -11808.922,E2 -11808.922} C_VEL
LIN {X 0,Y 390.029,Z 266.713,A -85,B 0,C 180,E1 -11812.234,E2 -11812.234} C_VEL
LIN {X 0,Y 390.107,Z 266.707,A -85,B 0,C 180,E1 -11815.743,E2 -11815.743} C_VEL
LIN {X 0,Y 390.047,Z 266.709,A -85,B 0,C 180,E1 -11819.11,E2 -11819.11} C_VEL
LIN {X 0,Y 390.033,Z 266.711,A -85,B 0,C 180,E1 -11820.815,E2 -11820.815} C_VEL
LIN {X 0,Y 389.362,Z 266.94,A -85,B 0,C 180,E1 -11821.181,E2 -11821.181} C_VEL
LIN {X 0,Y 386.686,Z 268.006,A -85,B 0,C 180,E1 -11821.692,E2 -11821.692} C_VEL
LIN {X 0,Y 384.075,Z 269.688,A -85,B 0,C 180,E1 -11822.187,E2 -11822.187} C_VEL
LIN {X 0,Y 383.537,Z 270.896,A -85,B 0,C 180,E1 -11822.525,E2 -11822.525} C_VEL
LIN {X 0,Y 383.545,Z 272.785,A -85,B 0,C 180,E1 -11823.056,E2 -11823.056} C_VEL
LIN {X 0,Y 386.61,Z 290.698,A -85,B 0,C 180,E1 -11823.554,E2 -11823.554} C_VEL
LIN {X 0,Y 385.757,Z 350.068,A -85,B 0,C 180,E1 -11824.77,E2 -11824.77} C_VEL
LIN {X 0,Y 385.489,Z 360.914,A -85,B 0,C 180,E1 -11825.162,E2 -11825.162} C_VEL
LIN {X 0,Y 385.126,Z 372.308,A -85,B 0,C 180,E1 -11825.799,E2 -11825.799} C_VEL
LIN {X 0,Y 384.695,Z 381.628,A -85,B 0,C 180,E1 -11826.504,E2 -11826.504} C_VEL
LIN {X 0,Y 384.332,Z 389.766,A -85,B 0,C 180,E1 -11827.28,E2 -11827.28} C_VEL
LIN {X 0,Y 383.833,Z 398.094,A -85,B 0,C 180,E1 -11828.258,E2 -11828.258} C_VEL
LIN {X 0,Y 383.268,Z 406.152,A -85,B 0,C 180,E1 -11829.428,E2 -11829.428} C_VEL
LIN {X 0,Y 382.85,Z 413.764,A -85,B 0,C 180,E1 -11830.855,E2 -11830.855} C_VEL
LIN {X 0,Y 382.434,Z 418.831,A -85,B 0,C 180,E1 -11832.038,E2 -11832.038} C_VEL
LIN {X 0,Y 382.319,Z 421.813,A -85,B 0,C 180,E1 -11832.854,E2 -11832.854} C_VEL
LIN {X 0,Y 382.07,Z 426.046,A -85,B 0,C 180,E1 -11834.345,E2 -11834.345} C_VEL
LIN {X 0,Y 381.772,Z 429.164,A -85,B 0,C 180,E1 -11835.884,E2 -11835.884} C_VEL
LIN {X 0,Y 381.624,Z 431.165,A -85,B 0,C 180,E1 -11837.444,E2 -11837.444} C_VEL
LIN {X 0,Y 381.601,Z 432.065,A -85,B 0,C 180,E1 -11839.033,E2 -11839.033} C_VEL
LIN {X 0,Y 381.681,Z 431.81,A -85,B 0,C 180,E1 -11840.655,E2 -11840.655} C_VEL
LIN {X 0,Y 381.948,Z 429.752,A -85,B 0,C 180,E1 -11842.613,E2 -11842.613} C_VEL
LIN {X 0,Y 382.196,Z 427.219,A -85,B 0,C 180,E1 -11844.005,E2 -11844.005} C_VEL
LIN {X 0,Y 382.508,Z 424.009,A -85,B 0,C 180,E1 -11845.281,E2 -11845.281} C_VEL
LIN {X 0,Y 382.871,Z 419.742,A -85,B 0,C 180,E1 -11846.588,E2 -11846.588} C_VEL
LIN {X 0,Y 383.314,Z 414.411,A -85,B 0,C 180,E1 -11847.88,E2 -11847.88} C_VEL
LIN {X 0,Y 383.975,Z 406.7,A -85,B 0,C 180,E1 -11849.343,E2 -11849.343} C_VEL
LIN {X 0,Y 384.622,Z 399.288,A -85,B 0,C 180,E1 -11850.44,E2 -11850.44} C_VEL
LIN {X 0,Y 385.197,Z 392.223,A -85,B 0,C 180,E1 -11851.302,E2 -11851.302} C_VEL
LIN {X 0,Y 385.721,Z 383.528,A -85,B 0,C 180,E1 -11852.168,E2 -11852.168} C_VEL
LIN {X 0,Y 386.155,Z 374.749,A -85,B 0,C 180,E1 -11852.863,E2 -11852.863} C_VEL
LIN {X 0,Y 386.67,Z 364.392,A -85,B 0,C 180,E1 -11853.486,E2 -11853.486} C_VEL
LIN {X 0,Y 386.956,Z 353.375,A -85,B 0,C 180,E1 -11853.942,E2 -11853.942} C_VEL
LIN {X 0,Y 387.225,Z 334.395,A -85,B 0,C 180,E1 -11854.377,E2 -11854.377} C_VEL
LIN {X 0,Y 387.906,Z 289.399,A -85,B 0,C 180,E1 -11855.303,E2 -11855.303} C_VEL
LIN {X 0,Y 384.637,Z 274.805,A -85,B 0,C 180,E1 -11855.798,E2 -11855.798} C_VEL
LIN {X 0,Y 384.128,Z 273.096,A -85,B 0,C 180,E1 -11855.908,E2 -11855.908} C_VEL
LIN {X 0,Y 383.015,Z 267.591,A -85,B 0,C 180,E1 -11857.337,E2 -11857.337} C_VEL
LIN {X 0,Y 383.05,Z 267.59,A -85,B 0,C 180,E1 -11860.717,E2 -11860.717} C_VEL
LIN {X 0,Y 383.07,Z 267.583,A -85,B 0,C 180,E1 -11864.027,E2 -11864.027} C_VEL
LIN {X 0,Y 383.127,Z 267.573,A -85,B 0,C 180,E1 -11867.285,E2 -11867.285} C_VEL
LIN {X 0,Y 383.142,Z 267.574,A -85,B 0,C 180,E1 -11870.499,E2 -11870.499} C_VEL
LIN {X 0,Y 383.281,Z 267.554,A -85,B 0,C 180,E1 -11873.685,E2 -11873.685} C_VEL
LIN {X 0,Y 383.379,Z 267.538,A -85,B 0,C 180,E1 -11877.9,E2 -11877.9} C_VEL
LIN {X 0,Y 383.51,Z 267.526,A -85,B 0,C 180,E1 -11880.001,E2 -11880.001} C_VEL
LIN {X 0,Y 383.244,Z 267.556,A -85,B 0,C 180,E1 -11883.155,E2 -11883.155} C_VEL
LIN {X 0,Y 383.279,Z 267.556,A -85,B 0,C 180,E1 -11886.317,E2 -11886.317} C_VEL
LIN {X 0,Y 383.252,Z 267.553,A -85,B 0,C 180,E1 -11888.437,E2 -11888.437} C_VEL
LIN {X 0,Y 383.089,Z 267.574,A -85,B 0,C 180,E1 -11891.643,E2 -11891.643} C_VEL
LIN {X 0,Y 383.103,Z 267.575,A -85,B 0,C 180,E1 -11894.883,E2 -11894.883} C_VEL
LIN {X 0,Y 383.082,Z 267.576,A -85,B 0,C 180,E1 -11898.173,E2 -11898.173} C_VEL
LIN {X 0,Y 382.987,Z 267.583,A -85,B 0,C 180,E1 -11901.532,E2 -11901.532} C_VEL
LIN {X 0,Y 383.046,Z 267.575,A -85,B 0,C 180,E1 -11904.961,E2 -11904.961} C_VEL
LIN {X 0,Y 383.044,Z 267.58,A -85,B 0,C 180,E1 -11908.493,E2 -11908.493} C_VEL
LIN {X 0,Y 383.006,Z 267.59,A -85,B 0,C 180,E1 -11912.151,E2 -11912.151} C_VEL
LIN {X 0,Y 383.014,Z 267.588,A -85,B 0,C 180,E1 -11914.669,E2 -11914.669} C_VEL
LIN {X 0,Y 382.999,Z 267.584,A -85,B 0,C 180,E1 -11917.906,E2 -11917.906} C_VEL
LIN {X 0,Y 383.01,Z 267.585,A -85,B 0,C 180,E1 -11921.345,E2 -11921.345} C_VEL
LIN {X 0,Y 382.993,Z 267.588,A -85,B 0,C 180,E1 -11924.304,E2 -11924.304} C_VEL
LIN {X 0,Y 383.008,Z 267.587,A -85,B 0,C 180,E1 -11927.241,E2 -11927.241} C_VEL
LIN {X 0,Y 383.014,Z 267.592,A -85,B 0,C 180,E1 -11930.414,E2 -11930.414} C_VEL
LIN {X 0,Y 383.025,Z 267.587,A -85,B 0,C 180,E1 -11934.046,E2 -11934.046} C_VEL
LIN {X 0,Y 382.986,Z 267.591,A -85,B 0,C 180,E1 -11937.579,E2 -11937.579} C_VEL
LIN {X 0,Y 382.992,Z 267.594,A -85,B 0,C 180,E1 -11940.301,E2 -11940.301} C_VEL
LIN {X 0,Y 383.094,Z 267.582,A -85,B 0,C 180,E1 -11943.145,E2 -11943.145} C_VEL
LIN {X 0,Y 385.145,Z 278.707,A -85,B 0,C 180,E1 -11945.838,E2 -11945.838} C_VEL
LIN {X 0,Y 384.814,Z 287.149,A -85,B 0,C 180,E1 -11947.731,E2 -11947.731} C_VEL
LIN {X 0,Y 383.675,Z 305.864,A -85,B 0,C 180,E1 -11951.857,E2 -11951.857} C_VEL
LIN {X 0,Y 383.342,Z 312.014,A -85,B 0,C 180,E1 -11953.149,E2 -11953.149} C_VEL
LIN {X 0,Y 386.251,Z 331.375,A -85,B 0,C 180,E1 -11953.719,E2 -11953.719} C_VEL
LIN {X 0,Y 387.384,Z 343.904,A -85,B 0,C 180,E1 -11954.041,E2 -11954.041} C_VEL
LIN {X 0,Y 386.609,Z 390.707,A -85,B 0,C 180,E1 -11955.019,E2 -11955.019} C_VEL
LIN {X 0,Y 386.165,Z 401.733,A -85,B 0,C 180,E1 -11955.408,E2 -11955.408} C_VEL
LIN {X 0,Y 385.493,Z 413.057,A -85,B 0,C 180,E1 -11956.022,E2 -11956.022} C_VEL
LIN {X 0,Y 384.744,Z 423.401,A -85,B 0,C 180,E1 -11956.802,E2 -11956.802} C_VEL
LIN {X 0,Y 384.114,Z 431.593,A -85,B 0,C 180,E1 -11957.586,E2 -11957.586} C_VEL
LIN {X 0,Y 383.499,Z 439.408,A -85,B 0,C 180,E1 -11958.505,E2 -11958.505} C_VEL
LIN {X 0,Y 382.895,Z 447.626,A -85,B 0,C 180,E1 -11959.691,E2 -11959.691} C_VEL
LIN {X 0,Y 382.335,Z 454.85,A -85,B 0,C 180,E1 -11961.011,E2 -11961.011} C_VEL
LIN {X 0,Y 382.081,Z 459.593,A -85,B 0,C 180,E1 -11962.071,E2 -11962.071} C_VEL
LIN {X 0,Y 381.86,Z 463.527,A -85,B 0,C 180,E1 -11963.13,E2 -11963.13} C_VEL
LIN {X 0,Y 381.686,Z 468.078,A -85,B 0,C 180,E1 -11964.718,E2 -11964.718} C_VEL
LIN {X 0,Y 381.687,Z 470.427,A -85,B 0,C 180,E1 -11965.777,E2 -11965.777} C_VEL
LIN {X 0,Y 381.635,Z 472.143,A -85,B 0,C 180,E1 -11966.833,E2 -11966.833} C_VEL
LIN {X 0,Y 381.726,Z 473.294,A -85,B 0,C 180,E1 -11967.89,E2 -11967.89} C_VEL
LIN {X 0,Y 381.714,Z 473.951,A -85,B 0,C 180,E1 -11968.945,E2 -11968.945} C_VEL
LIN {X 0,Y 381.721,Z 474.13,A -85,B 0,C 180,E1 -11970,E2 -11970} C_VEL
LIN {X 0,Y 381.722,Z 473.806,A -85,B 0,C 180,E1 -11971.055,E2 -11971.055} C_VEL
LIN {X 0,Y 381.75,Z 472.875,A -85,B 0,C 180,E1 -11972.11,E2 -11972.11} C_VEL
LIN {X 0,Y 381.672,Z 471.401,A -85,B 0,C 180,E1 -11973.167,E2 -11973.167} C_VEL
LIN {X 0,Y 381.752,Z 468.24,A -85,B 0,C 180,E1 -11974.752,E2 -11974.752} C_VEL
LIN {X 0,Y 381.769,Z 463.63,A -85,B 0,C 180,E1 -11976.342,E2 -11976.342} C_VEL
LIN {X 0,Y 382.007,Z 458.527,A -85,B 0,C 180,E1 -11977.665,E2 -11977.665} C_VEL
LIN {X 0,Y 382.23,Z 453.536,A -85,B 0,C 180,E1 -11978.725,E2 -11978.725} C_VEL
LIN {X 0,Y 382.568,Z 447.515,A -85,B 0,C 180,E1 -11979.784,E2 -11979.784} C_VEL
LIN {X 0,Y 383.029,Z 440.184,A -85,B 0,C 180,E1 -11980.84,E2 -11980.84} C_VEL
LIN {X 0,Y 383.487,Z 432.348,A -85,B 0,C 180,E1 -11981.764,E2 -11981.764} C_VEL
LIN {X 0,Y 383.993,Z 424.11,A -85,B 0,C 180,E1 -11982.553,E2 -11982.553} C_VEL
LIN {X 0,Y 384.577,Z 413.681,A -85,B 0,C 180,E1 -11983.339,E2 -11983.339} C_VEL
LIN {X 0,Y 385.134,Z 401.987,A -85,B 0,C 180,E1 -11983.958,E2 -11983.958} C_VEL
LIN {X 0,Y 385.512,Z 392.992,A -85,B 0,C 180,E1 -11984.281,E2 -11984.281} C_VEL
LIN {X 0,Y 385.914,Z 364.747,A -85,B 0,C 180,E1 -11984.879,E2 -11984.879} C_VEL
LIN {X 0,Y 386.028,Z 340.142,A -85,B 0,C 180,E1 -11985.379,E2 -11985.379} C_VEL
LIN {X 0,Y 383.048,Z 313.712,A -85,B 0,C 180,E1 -11986.043,E2 -11986.043} C_VEL
LIN {X 0,Y 383.894,Z 298.562,A -85,B 0,C 180,E1 -11989.518,E2 -11989.518} C_VEL
LIN {X 0,Y 385.096,Z 281.859,A -85,B 0,C 180,E1 -11993.387,E2 -11993.387} C_VEL
LIN {X 0,Y 384.875,Z 277.534,A -85,B 0,C 180,E1 -11994.423,E2 -11994.423} C_VEL
LIN {X 0,Y 383.121,Z 267.576,A -85,B 0,C 180,E1 -11996.927,E2 -11996.927} C_VEL
LIN {X 0,Y 382.984,Z 267.588,A -85,B 0,C 180,E1 -12000.918,E2 -12000.918} C_VEL
LIN {X 0,Y 383.019,Z 267.583,A -85,B 0,C 180,E1 -12004.667,E2 -12004.667} C_VEL
LIN {X 0,Y 383,Z 267.588,A -85,B 0,C 180,E1 -12007.903,E2 -12007.903} C_VEL
LIN {X 0,Y 382.984,Z 267.592,A -85,B 0,C 180,E1 -12011.347,E2 -12011.347} C_VEL
LIN {X 0,Y 382.995,Z 267.587,A -85,B 0,C 180,E1 -12014.303,E2 -12014.303} C_VEL
LIN {X 0,Y 383.01,Z 267.588,A -85,B 0,C 180,E1 -12017.239,E2 -12017.239} C_VEL
LIN {X 0,Y 383.012,Z 267.584,A -85,B 0,C 180,E1 -12020.413,E2 -12020.413} C_VEL
LIN {X 0,Y 383.023,Z 267.585,A -85,B 0,C 180,E1 -12024.044,E2 -12024.044} C_VEL
LIN {X 0,Y 383.003,Z 267.592,A -85,B 0,C 180,E1 -12027.573,E2 -12027.573} C_VEL
LIN {X 0,Y 382.989,Z 267.588,A -85,B 0,C 180,E1 -12030.299,E2 -12030.299} C_VEL
LIN {X 0,Y 383.054,Z 267.579,A -85,B 0,C 180,E1 -12032.697,E2 -12032.697} C_VEL
LIN {X 0,Y 383.031,Z 267.583,A -85,B 0,C 180,E1 -12036.192,E2 -12036.192} C_VEL
LIN {X 0,Y 383.052,Z 267.586,A -85,B 0,C 180,E1 -12039.598,E2 -12039.598} C_VEL
LIN {X 0,Y 383.101,Z 267.574,A -85,B 0,C 180,E1 -12042.93,E2 -12042.93} C_VEL
LIN {X 0,Y 383.121,Z 267.571,A -85,B 0,C 180,E1 -12046.463,E2 -12046.463} C_VEL
LIN {X 0,Y 383.147,Z 267.568,A -85,B 0,C 180,E1 -12050.497,E2 -12050.497} C_VEL
LIN {X 0,Y 383.278,Z 267.557,A -85,B 0,C 180,E1 -12053.683,E2 -12053.683} C_VEL
LIN {X 0,Y 383.382,Z 267.542,A -85,B 0,C 180,E1 -12057.898,E2 -12057.898} C_VEL
LIN {X 0,Y 383.514,Z 267.524,A -85,B 0,C 180,E1 -12059.999,E2 -12059.999} C_VEL
LIN {X 0,Y 383.246,Z 267.557,A -85,B 0,C 180,E1 -12063.153,E2 -12063.153} C_VEL
LIN {X 0,Y 383.262,Z 267.553,A -85,B 0,C 180,E1 -12066.648,E2 -12066.648} C_VEL
LIN {X 0,Y 383.255,Z 267.554,A -85,B 0,C 180,E1 -12068.435,E2 -12068.435} C_VEL
LIN {X 0,Y 383.101,Z 267.58,A -85,B 0,C 180,E1 -12071.641,E2 -12071.641} C_VEL
LIN {X 0,Y 383.105,Z 267.573,A -85,B 0,C 180,E1 -12074.881,E2 -12074.881} C_VEL
LIN {X 0,Y 383.086,Z 267.577,A -85,B 0,C 180,E1 -12078.171,E2 -12078.171} C_VEL
LIN {X 0,Y 382.997,Z 267.591,A -85,B 0,C 180,E1 -12081.53,E2 -12081.53} C_VEL
LIN {X 0,Y 383.044,Z 267.581,A -85,B 0,C 180,E1 -12084.96,E2 -12084.96} C_VEL
LIN {X 0,Y 383.021,Z 267.585,A -85,B 0,C 180,E1 -12088.269,E2 -12088.269} C_VEL
LIN {X 0,Y 383.001,Z 267.588,A -85,B 0,C 180,E1 -12092.149,E2 -12092.149} C_VEL
LIN {X 0,Y 383.01,Z 267.585,A -85,B 0,C 180,E1 -12094.667,E2 -12094.667} C_VEL
LIN {X 0,Y 382.995,Z 267.59,A -85,B 0,C 180,E1 -12097.904,E2 -12097.904} C_VEL
LIN {X 0,Y 383.006,Z 267.588,A -85,B 0,C 180,E1 -12101.343,E2 -12101.343} C_VEL
LIN {X 0,Y 383.001,Z 267.587,A -85,B 0,C 180,E1 -12104.305,E2 -12104.305} C_VEL
LIN {X 0,Y 383.067,Z 267.58,A -85,B 0,C 180,E1 -12107.249,E2 -12107.249} C_VEL
LIN {X 0,Y 383.013,Z 267.585,A -85,B 0,C 180,E1 -12110.412,E2 -12110.412} C_VEL
LIN {X 0,Y 383.018,Z 267.587,A -85,B 0,C 180,E1 -12114.044,E2 -12114.044} C_VEL
LIN {X 0,Y 382.978,Z 267.594,A -85,B 0,C 180,E1 -12117.578,E2 -12117.578} C_VEL
LIN {X 0,Y 382.983,Z 267.59,A -85,B 0,C 180,E1 -12120.3,E2 -12120.3} C_VEL
LIN {X 0,Y 383.048,Z 267.58,A -85,B 0,C 180,E1 -12122.698,E2 -12122.698} C_VEL
LIN {X 0,Y 383.025,Z 267.585,A -85,B 0,C 180,E1 -12126.192,E2 -12126.192} C_VEL
LIN {X 0,Y 383.052,Z 267.585,A -85,B 0,C 180,E1 -12129.598,E2 -12129.598} C_VEL
LIN {X 0,Y 383.096,Z 267.574,A -85,B 0,C 180,E1 -12132.931,E2 -12132.931} C_VEL
LIN {X 0,Y 383.117,Z 267.572,A -85,B 0,C 180,E1 -12136.464,E2 -12136.464} C_VEL
LIN {X 0,Y 383.143,Z 267.569,A -85,B 0,C 180,E1 -12140.498,E2 -12140.498} C_VEL
LIN {X 0,Y 383.263,Z 267.554,A -85,B 0,C 180,E1 -12142.625,E2 -12142.625} C_VEL
LIN {X 0,Y 383.187,Z 267.563,A -85,B 0,C 180,E1 -12144.738,E2 -12144.738} C_VEL
LIN {X 0,Y 383.376,Z 267.544,A -85,B 0,C 180,E1 -12147.899,E2 -12147.899} C_VEL
LIN {X 0,Y 383.51,Z 267.526,A -85,B 0,C 180,E1 -12150,E2 -12150} C_VEL
LIN {X 0,Y 383.237,Z 267.558,A -85,B 0,C 180,E1 -12153.153,E2 -12153.153} C_VEL
LIN {X 0,Y 383.27,Z 267.554,A -85,B 0,C 180,E1 -12156.316,E2 -12156.316} C_VEL
LIN {X 0,Y 383.147,Z 267.571,A -85,B 0,C 180,E1 -12159.502,E2 -12159.502} C_VEL
LIN {X 0,Y 383.132,Z 267.57,A -85,B 0,C 180,E1 -12162.716,E2 -12162.716} C_VEL
LIN {X 0,Y 383.071,Z 267.581,A -85,B 0,C 180,E1 -12165.973,E2 -12165.973} C_VEL
LIN {X 0,Y 383.05,Z 267.582,A -85,B 0,C 180,E1 -12169.284,E2 -12169.284} C_VEL
LIN {X 0,Y 382.986,Z 267.588,A -85,B 0,C 180,E1 -12172.665,E2 -12172.665} C_VEL
LIN {X 0,Y 383.068,Z 267.581,A -85,B 0,C 180,E1 -12176.123,E2 -12176.123} C_VEL
LIN {X 0,Y 382.993,Z 267.592,A -85,B 0,C 180,E1 -12179.699,E2 -12179.699} C_VEL
LIN {X 0,Y 383.087,Z 267.697,A -85,B 0,C 180,E1 -12181.6,E2 -12181.6} C_VEL
LIN {X 0,Y 383.537,Z 270.896,A -85,B 0,C 180,E1 -12182.525,E2 -12182.525} C_VEL
LIN {X 0,Y 383.097,Z 272.664,A -85,B 0,C 180,E1 -12182.816,E2 -12182.816} C_VEL
LIN {X 0,Y 381.45,Z 275.756,A -85,B 0,C 180,E1 -12183.015,E2 -12183.015} C_VEL
LIN {X 0,Y 378.003,Z 282.181,A -85,B 0,C 180,E1 -12183.059,E2 -12183.059} C_VEL
LIN {X 0,Y 377.2,Z 286.404,A -85,B 0,C 180,E1 -12183.108,E2 -12183.108} C_VEL
LIN {X 0,Y 377.594,Z 290.793,A -85,B 0,C 180,E1 -12183.211,E2 -12183.211} C_VEL
LIN {X 0,Y 379.502,Z 300.616,A -85,B 0,C 180,E1 -12183.503,E2 -12183.503} C_VEL
LIN {X 0,Y 379.551,Z 301.735,A -85,B 0,C 180,E1 -12183.529,E2 -12183.529} C_VEL
LIN {X 0,Y 378.831,Z 349.96,A -85,B 0,C 180,E1 -12184.539,E2 -12184.539} C_VEL
LIN {X 0,Y 378.547,Z 360.371,A -85,B 0,C 180,E1 -12184.913,E2 -12184.913} C_VEL
LIN {X 0,Y 378.154,Z 372.747,A -85,B 0,C 180,E1 -12185.604,E2 -12185.604} C_VEL
LIN {X 0,Y 377.753,Z 381.386,A -85,B 0,C 180,E1 -12186.263,E2 -12186.263} C_VEL
LIN {X 0,Y 377.387,Z 389.513,A -85,B 0,C 180,E1 -12187.04,E2 -12187.04} C_VEL
LIN {X 0,Y 376.891,Z 397.494,A -85,B 0,C 180,E1 -12187.977,E2 -12187.977} C_VEL
LIN {X 0,Y 376.413,Z 403.899,A -85,B 0,C 180,E1 -12188.884,E2 -12188.884} C_VEL
LIN {X 0,Y 376.012,Z 410.295,A -85,B 0,C 180,E1 -12189.977,E2 -12189.977} C_VEL
LIN {X 0,Y 375.641,Z 416.196,A -85,B 0,C 180,E1 -12191.207,E2 -12191.207} C_VEL
LIN {X 0,Y 375.273,Z 421.99,A -85,B 0,C 180,E1 -12192.721,E2 -12192.721} C_VEL
LIN {X 0,Y 375.034,Z 425.444,A -85,B 0,C 180,E1 -12193.896,E2 -12193.896} C_VEL
LIN {X 0,Y 374.763,Z 428.893,A -85,B 0,C 180,E1 -12195.447,E2 -12195.447} C_VEL
LIN {X 0,Y 374.531,Z 431.605,A -85,B 0,C 180,E1 -12197.506,E2 -12197.506} C_VEL
LIN {X 0,Y 374.529,Z 432.416,A -85,B 0,C 180,E1 -12198.948,E2 -12198.948} C_VEL
LIN {X 0,Y 374.598,Z 432.321,A -85,B 0,C 180,E1 -12200.367,E2 -12200.367} C_VEL
LIN {X 0,Y 374.737,Z 431.186,A -85,B 0,C 180,E1 -12201.968,E2 -12201.968} C_VEL
LIN {X 0,Y 375.057,Z 428.612,A -85,B 0,C 180,E1 -12203.681,E2 -12203.681} C_VEL
LIN {X 0,Y 375.379,Z 425.613,A -85,B 0,C 180,E1 -12205.018,E2 -12205.018} C_VEL
LIN {X 0,Y 375.809,Z 421.056,A -85,B 0,C 180,E1 -12206.519,E2 -12206.519} C_VEL
LIN {X 0,Y 376.165,Z 417.148,A -85,B 0,C 180,E1 -12207.554,E2 -12207.554} C_VEL
LIN {X 0,Y 376.69,Z 411.15,A -85,B 0,C 180,E1 -12208.84,E2 -12208.84} C_VEL
LIN {X 0,Y 377.165,Z 405.751,A -85,B 0,C 180,E1 -12209.795,E2 -12209.795} C_VEL
LIN {X 0,Y 377.757,Z 399.467,A -85,B 0,C 180,E1 -12210.727,E2 -12210.727} C_VEL
LIN {X 0,Y 378.352,Z 392.591,A -85,B 0,C 180,E1 -12211.577,E2 -12211.577} C_VEL
LIN {X 0,Y 378.843,Z 384.868,A -85,B 0,C 180,E1 -12212.37,E2 -12212.37} C_VEL
LIN {X 0,Y 379.314,Z 375.864,A -85,B 0,C 180,E1 -12213.11,E2 -12213.11} C_VEL
LIN {X 0,Y 379.775,Z 367.651,A -85,B 0,C 180,E1 -12213.633,E2 -12213.633} C_VEL
LIN {X 0,Y 380.029,Z 358.527,A -85,B 0,C 180,E1 -12214.078,E2 -12214.078} C_VEL
LIN {X 0,Y 380.278,Z 348.054,A -85,B 0,C 180,E1 -12214.418,E2 -12214.418} C_VEL
LIN {X 0,Y 381.261,Z 290.548,A -85,B 0,C 180,E1 -12215.638,E2 -12215.638} C_VEL
LIN {X 0,Y 378.354,Z 277.454,A -85,B 0,C 180,E1 -12216.096,E2 -12216.096} C_VEL
LIN {X 0,Y 377.055,Z 273.556,A -85,B 0,C 180,E1 -12216.292,E2 -12216.292} C_VEL
LIN {X 0,Y 375.963,Z 268.47,A -85,B 0,C 180,E1 -12217.686,E2 -12217.686} C_VEL
LIN {X 0,Y 375.987,Z 268.471,A -85,B 0,C 180,E1 -12220.34,E2 -12220.34} C_VEL
LIN {X 0,Y 376.018,Z 268.46,A -85,B 0,C 180,E1 -12223.72,E2 -12223.72} C_VEL
LIN {X 0,Y 376.094,Z 268.45,A -85,B 0,C 180,E1 -12227.043,E2 -12227.043} C_VEL
LIN {X 0,Y 376.11,Z 268.448,A -85,B 0,C 180,E1 -12230.319,E2 -12230.319} C_VEL
LIN {X 0,Y 376.238,Z 268.431,A -85,B 0,C 180,E1 -12233.566,E2 -12233.566} C_VEL
LIN {X 0,Y 376.345,Z 268.414,A -85,B 0,C 180,E1 -12237.861,E2 -12237.861} C_VEL
LIN {X 0,Y 376.48,Z 268.402,A -85,B 0,C 180,E1 -12240.001,E2 -12240.001} C_VEL
LIN {X 0,Y 376.182,Z 268.436,A -85,B 0,C 180,E1 -12243.214,E2 -12243.214} C_VEL
LIN {X 0,Y 376.238,Z 268.434,A -85,B 0,C 180,E1 -12246.436,E2 -12246.436} C_VEL
LIN {X 0,Y 376.198,Z 268.432,A -85,B 0,C 180,E1 -12248.596,E2 -12248.596} C_VEL
LIN {X 0,Y 376.042,Z 268.453,A -85,B 0,C 180,E1 -12251.864,E2 -12251.864} C_VEL
LIN {X 0,Y 376.051,Z 268.452,A -85,B 0,C 180,E1 -12255.168,E2 -12255.168} C_VEL
LIN {X 0,Y 376.017,Z 268.46,A -85,B 0,C 180,E1 -12258.527,E2 -12258.527} C_VEL
LIN {X 0,Y 375.957,Z 268.46,A -85,B 0,C 180,E1 -12261.955,E2 -12261.955} C_VEL
LIN {X 0,Y 376,Z 268.452,A -85,B 0,C 180,E1 -12265.462,E2 -12265.462} C_VEL
LIN {X 0,Y 375.971,Z 268.456,A -85,B 0,C 180,E1 -12269.08,E2 -12269.08} C_VEL
LIN {X 0,Y 375.945,Z 268.462,A -85,B 0,C 180,E1 -12272.83,E2 -12272.83} C_VEL
LIN {X 0,Y 375.954,Z 268.465,A -85,B 0,C 180,E1 -12275.417,E2 -12275.417} C_VEL
LIN {X 0,Y 375.974,Z 268.462,A -85,B 0,C 180,E1 -12278.272,E2 -12278.272} C_VEL
LIN {X 0,Y 375.957,Z 268.464,A -85,B 0,C 180,E1 -12281.606,E2 -12281.606} C_VEL
LIN {X 0,Y 375.924,Z 268.47,A -85,B 0,C 180,E1 -12285.27,E2 -12285.27} C_VEL
LIN {X 0,Y 375.932,Z 268.472,A -85,B 0,C 180,E1 -12288.4,E2 -12288.4} C_VEL
LIN {X 0,Y 375.974,Z 268.463,A -85,B 0,C 180,E1 -12291.73,E2 -12291.73} C_VEL
LIN {X 0,Y 375.979,Z 268.464,A -85,B 0,C 180,E1 -12295.334,E2 -12295.334} C_VEL
LIN {X 0,Y 375.957,Z 268.47,A -85,B 0,C 180,E1 -12298.439,E2 -12298.439} C_VEL
LIN {X 0,Y 375.989,Z 268.467,A -85,B 0,C 180,E1 -12302.142,E2 -12302.142} C_VEL
LIN {X 0,Y 376.046,Z 268.571,A -85,B 0,C 180,E1 -12302.863,E2 -12302.863} C_VEL
LIN {X 0,Y 377.916,Z 278.191,A -85,B 0,C 180,E1 -12305.27,E2 -12305.27} C_VEL
LIN {X 0,Y 378.278,Z 281.944,A -85,B 0,C 180,E1 -12306.167,E2 -12306.167} C_VEL
LIN {X 0,Y 377.246,Z 296.958,A -85,B 0,C 180,E1 -12309.556,E2 -12309.556} C_VEL
LIN {X 0,Y 376.403,Z 311.218,A -85,B 0,C 180,E1 -12312.741,E2 -12312.741} C_VEL
LIN {X 0,Y 379.432,Z 331.142,A -85,B 0,C 180,E1 -12313.365,E2 -12313.365} C_VEL
LIN {X 0,Y 380.631,Z 343.957,A -85,B 0,C 180,E1 -12313.708,E2 -12313.708} C_VEL
LIN {X 0,Y 379.812,Z 390.098,A -85,B 0,C 180,E1 -12314.691,E2 -12314.691} C_VEL
LIN {X 0,Y 379.406,Z 400.803,A -85,B 0,C 180,E1 -12315.073,E2 -12315.073} C_VEL
LIN {X 0,Y 378.635,Z 413.273,A -85,B 0,C 180,E1 -12315.763,E2 -12315.763} C_VEL
LIN {X 0,Y 377.974,Z 421.989,A -85,B 0,C 180,E1 -12316.424,E2 -12316.424} C_VEL
LIN {X 0,Y 377.309,Z 430.358,A -85,B 0,C 180,E1 -12317.222,E2 -12317.222} C_VEL
LIN {X 0,Y 376.589,Z 438.311,A -85,B 0,C 180,E1 -12318.154,E2 -12318.154} C_VEL
LIN {X 0,Y 376.04,Z 445.777,A -85,B 0,C 180,E1 -12319.229,E2 -12319.229} C_VEL
LIN {X 0,Y 375.433,Z 453.375,A -85,B 0,C 180,E1 -12320.573,E2 -12320.573} C_VEL
LIN {X 0,Y 375.023,Z 459.346,A -85,B 0,C 180,E1 -12321.921,E2 -12321.921} C_VEL
LIN {X 0,Y 374.802,Z 463.259,A -85,B 0,C 180,E1 -12323,E2 -12323} C_VEL
LIN {X 0,Y 374.591,Z 467.762,A -85,B 0,C 180,E1 -12324.618,E2 -12324.618} C_VEL
LIN {X 0,Y 374.616,Z 470.09,A -85,B 0,C 180,E1 -12325.697,E2 -12325.697} C_VEL
LIN {X 0,Y 374.545,Z 471.802,A -85,B 0,C 180,E1 -12326.773,E2 -12326.773} C_VEL
LIN {X 0,Y 374.626,Z 472.933,A -85,B 0,C 180,E1 -12327.85,E2 -12327.85} C_VEL
LIN {X 0,Y 374.646,Z 473.568,A -85,B 0,C 180,E1 -12328.925,E2 -12328.925} C_VEL
LIN {X 0,Y 374.651,Z 473.721,A -85,B 0,C 180,E1 -12330,E2 -12330} C_VEL
LIN {X 0,Y 374.654,Z 473.382,A -85,B 0,C 180,E1 -12331.075,E2 -12331.075} C_VEL
LIN {X 0,Y 374.666,Z 472.442,A -85,B 0,C 180,E1 -12332.15,E2 -12332.15} C_VEL
LIN {X 0,Y 374.585,Z 470.068,A -85,B 0,C 180,E1 -12333.765,E2 -12333.765} C_VEL
LIN {X 0,Y 374.618,Z 466.308,A -85,B 0,C 180,E1 -12335.383,E2 -12335.383} C_VEL
LIN {X 0,Y 374.714,Z 463.071,A -85,B 0,C 180,E1 -12336.462,E2 -12336.462} C_VEL
LIN {X 0,Y 374.94,Z 457.925,A -85,B 0,C 180,E1 -12337.811,E2 -12337.811} C_VEL
LIN {X 0,Y 375.202,Z 452.891,A -85,B 0,C 180,E1 -12338.89,E2 -12338.89} C_VEL
LIN {X 0,Y 375.537,Z 446.814,A -85,B 0,C 180,E1 -12339.969,E2 -12339.969} C_VEL
LIN {X 0,Y 376.023,Z 439.418,A -85,B 0,C 180,E1 -12341.045,E2 -12341.045} C_VEL
LIN {X 0,Y 376.518,Z 431.506,A -85,B 0,C 180,E1 -12341.985,E2 -12341.985} C_VEL
LIN {X 0,Y 377.047,Z 423.169,A -85,B 0,C 180,E1 -12342.788,E2 -12342.788} C_VEL
LIN {X 0,Y 377.631,Z 412.572,A -85,B 0,C 180,E1 -12343.589,E2 -12343.589} C_VEL
LIN {X 0,Y 378.171,Z 401.209,A -85,B 0,C 180,E1 -12344.186,E2 -12344.186} C_VEL
LIN {X 0,Y 378.571,Z 392.025,A -85,B 0,C 180,E1 -12344.514,E2 -12344.514} C_VEL
LIN {X 0,Y 379.203,Z 341.651,A -85,B 0,C 180,E1 -12345.578,E2 -12345.578} C_VEL
LIN {X 0,Y 376.045,Z 313.283,A -85,B 0,C 180,E1 -12346.315,E2 -12346.315} C_VEL
LIN {X 0,Y 377.048,Z 296.816,A -85,B 0,C 180,E1 -12350.171,E2 -12350.171} C_VEL
LIN {X 0,Y 378.159,Z 281.281,A -85,B 0,C 180,E1 -12353.842,E2 -12353.842} C_VEL
LIN {X 0,Y 376.891,Z 272.865,A -85,B 0,C 180,E1 -12355.956,E2 -12355.956} C_VEL
LIN {X 0,Y 376.053,Z 268.456,A -85,B 0,C 180,E1 -12357.099,E2 -12357.099} C_VEL
LIN {X 0,Y 375.957,Z 268.463,A -85,B 0,C 180,E1 -12360.693,E2 -12360.693} C_VEL
LIN {X 0,Y 375.961,Z 268.464,A -85,B 0,C 180,E1 -12364.111,E2 -12364.111} C_VEL
LIN {X 0,Y 375.954,Z 268.463,A -85,B 0,C 180,E1 -12366.741,E2 -12366.741} C_VEL
LIN {X 0,Y 375.989,Z 268.461,A -85,B 0,C 180,E1 -12369.97,E2 -12369.97} C_VEL
LIN {X 0,Y 375.93,Z 268.471,A -85,B 0,C 180,E1 -12373.765,E2 -12373.765} C_VEL
LIN {X 0,Y 375.933,Z 268.466,A -85,B 0,C 180,E1 -12376.81,E2 -12376.81} C_VEL
LIN {X 0,Y 375.959,Z 268.463,A -85,B 0,C 180,E1 -12380.536,E2 -12380.536} C_VEL
LIN {X 0,Y 375.962,Z 268.468,A -85,B 0,C 180,E1 -12383.495,E2 -12383.495} C_VEL
LIN {X 0,Y 375.958,Z 268.466,A -85,B 0,C 180,E1 -12385.888,E2 -12385.888} C_VEL
LIN {X 0,Y 375.962,Z 268.468,A -85,B 0,C 180,E1 -12389.686,E2 -12389.686} C_VEL
LIN {X 0,Y 375.994,Z 268.46,A -85,B 0,C 180,E1 -12392.14,E2 -12392.14} C_VEL
LIN {X 0,Y 376.004,Z 268.457,A -85,B 0,C 180,E1 -12394.538,E2 -12394.538} C_VEL
LIN {X 0,Y 375.96,Z 268.465,A -85,B 0,C 180,E1 -12398.045,E2 -12398.045} C_VEL
LIN {X 0,Y 376.02,Z 268.46,A -85,B 0,C 180,E1 -12401.473,E2 -12401.473} C_VEL
LIN {X 0,Y 376.054,Z 268.451,A -85,B 0,C 180,E1 -12404.832,E2 -12404.832} C_VEL
LIN {X 0,Y 376.045,Z 268.454,A -85,B 0,C 180,E1 -12408.136,E2 -12408.136} C_VEL
LIN {X 0,Y 376.215,Z 268.434,A -85,B 0,C 180,E1 -12411.918,E2 -12411.918} C_VEL
LIN {X 0,Y 376.166,Z 268.437,A -85,B 0,C 180,E1 -12414.639,E2 -12414.639} C_VEL
LIN {X 0,Y 376.348,Z 268.418,A -85,B 0,C 180,E1 -12417.859,E2 -12417.859} C_VEL
LIN {X 0,Y 376.483,Z 268.4,A -85,B 0,C 180,E1 -12419.999,E2 -12419.999} C_VEL
LIN {X 0,Y 376.184,Z 268.437,A -85,B 0,C 180,E1 -12423.212,E2 -12423.212} C_VEL
LIN {X 0,Y 376.227,Z 268.43,A -85,B 0,C 180,E1 -12426.64,E2 -12426.64} C_VEL
LIN {X 0,Y 376.2,Z 268.433,A -85,B 0,C 180,E1 -12428.594,E2 -12428.594} C_VEL
LIN {X 0,Y 376.052,Z 268.455,A -85,B 0,C 180,E1 -12431.862,E2 -12431.862} C_VEL
LIN {X 0,Y 376.053,Z 268.453,A -85,B 0,C 180,E1 -12435.167,E2 -12435.167} C_VEL
LIN {X 0,Y 376.023,Z 268.455,A -85,B 0,C 180,E1 -12438.525,E2 -12438.525} C_VEL
LIN {X 0,Y 375.963,Z 268.466,A -85,B 0,C 180,E1 -12441.953,E2 -12441.953} C_VEL
LIN {X 0,Y 375.999,Z 268.462,A -85,B 0,C 180,E1 -12445.46,E2 -12445.46} C_VEL
LIN {X 0,Y 375.953,Z 268.465,A -85,B 0,C 180,E1 -12449.079,E2 -12449.079} C_VEL
LIN {X 0,Y 375.941,Z 268.465,A -85,B 0,C 180,E1 -12452.828,E2 -12452.828} C_VEL
LIN {X 0,Y 375.95,Z 268.468,A -85,B 0,C 180,E1 -12455.415,E2 -12455.415} C_VEL
LIN {X 0,Y 375.969,Z 268.463,A -85,B 0,C 180,E1 -12458.271,E2 -12458.271} C_VEL
LIN {X 0,Y 375.952,Z 268.469,A -85,B 0,C 180,E1 -12461.605,E2 -12461.605} C_VEL
LIN {X 0,Y 375.971,Z 268.464,A -85,B 0,C 180,E1 -12465.26,E2 -12465.26} C_VEL
LIN {X 0,Y 375.981,Z 268.461,A -85,B 0,C 180,E1 -12468.389,E2 -12468.389} C_VEL
LIN {X 0,Y 375.959,Z 268.467,A -85,B 0,C 180,E1 -12471.911,E2 -12471.911} C_VEL
LIN {X 0,Y 375.971,Z 268.464,A -85,B 0,C 180,E1 -12475.332,E2 -12475.332} C_VEL
LIN {X 0,Y 375.949,Z 268.465,A -85,B 0,C 180,E1 -12478.438,E2 -12478.438} C_VEL
LIN {X 0,Y 375.987,Z 268.462,A -85,B 0,C 180,E1 -12482.141,E2 -12482.141} C_VEL
LIN {X 0,Y 375.998,Z 268.459,A -85,B 0,C 180,E1 -12484.539,E2 -12484.539} C_VEL
LIN {X 0,Y 375.957,Z 268.466,A -85,B 0,C 180,E1 -12488.046,E2 -12488.046} C_VEL
LIN {X 0,Y 376.016,Z 268.46,A -85,B 0,C 180,E1 -12491.474,E2 -12491.474} C_VEL
LIN {X 0,Y 376.05,Z 268.452,A -85,B 0,C 180,E1 -12494.832,E2 -12494.832} C_VEL
LIN {X 0,Y 376.042,Z 268.455,A -85,B 0,C 180,E1 -12498.136,E2 -12498.136} C_VEL
LIN {X 0,Y 376.248,Z 268.432,A -85,B 0,C 180,E1 -12501.878,E2 -12501.878} C_VEL
LIN {X 0,Y 376.16,Z 268.438,A -85,B 0,C 180,E1 -12504.64,E2 -12504.64} C_VEL
LIN {X 0,Y 376.342,Z 268.42,A -85,B 0,C 180,E1 -12507.859,E2 -12507.859} C_VEL
LIN {X 0,Y 376.479,Z 268.402,A -85,B 0,C 180,E1 -12510,E2 -12510} C_VEL
LIN {X 0,Y 376.175,Z 268.438,A -85,B 0,C 180,E1 -12513.213,E2 -12513.213} C_VEL
LIN {X 0,Y 376.229,Z 268.431,A -85,B 0,C 180,E1 -12516.435,E2 -12516.435} C_VEL
LIN {X 0,Y 376.114,Z 268.449,A -85,B 0,C 180,E1 -12519.681,E2 -12519.681} C_VEL
LIN {X 0,Y 376.08,Z 268.453,A -85,B 0,C 180,E1 -12523.658,E2 -12523.658} C_VEL
LIN {X 0,Y 376.033,Z 268.458,A -85,B 0,C 180,E1 -12527.607,E2 -12527.607} C_VEL
LIN {X 0,Y 375.968,Z 268.462,A -85,B 0,C 180,E1 -12530.832,E2 -12530.832} C_VEL
LIN {X 0,Y 375.979,Z 268.463,A -85,B 0,C 180,E1 -12534.282,E2 -12534.282} C_VEL
LIN {X 0,Y 376.009,Z 268.458,A -85,B 0,C 180,E1 -12536.652,E2 -12536.652} C_VEL
LIN {X 0,Y 375.959,Z 268.465,A -85,B 0,C 180,E1 -12540.312,E2 -12540.312} C_VEL
LIN {X 0,Y 376.03,Z 268.639,A -85,B 0,C 180,E1 -12541.488,E2 -12541.488} C_VEL
LIN {X 0,Y 376.557,Z 273.178,A -85,B 0,C 180,E1 -12542.808,E2 -12542.808} C_VEL
LIN {X 0,Y 379.728,Z 291.001,A -85,B 0,C 180,E1 -12543.309,E2 -12543.309} C_VEL
LIN {X 0,Y 379.551,Z 301.735,A -85,B 0,C 180,E1 -12543.529,E2 -12543.529} C_VEL
LIN {X 0,Y 378.926,Z 307.561,A -85,B 0,C 180,E1 -12543.629,E2 -12543.629} C_VEL
LIN {X 0,Y 372.952,Z 326.459,A -85,B 0,C 180,E1 -12543.822,E2 -12543.822} C_VEL
LIN {X 0,Y 372.124,Z 332.295,A -85,B 0,C 180,E1 -12543.917,E2 -12543.917} C_VEL
LIN {X 0,Y 371.849,Z 352.189,A -85,B 0,C 180,E1 -12544.375,E2 -12544.375} C_VEL
LIN {X 0,Y 371.538,Z 364.572,A -85,B 0,C 180,E1 -12544.894,E2 -12544.894} C_VEL
LIN {X 0,Y 371.128,Z 374.178,A -85,B 0,C 180,E1 -12545.486,E2 -12545.486} C_VEL
LIN {X 0,Y 370.73,Z 382.625,A -85,B 0,C 180,E1 -12546.159,E2 -12546.159} C_VEL
LIN {X 0,Y 370.367,Z 390.298,A -85,B 0,C 180,E1 -12546.917,E2 -12546.917} C_VEL
LIN {X 0,Y 369.906,Z 397.571,A -85,B 0,C 180,E1 -12547.786,E2 -12547.786} C_VEL
LIN {X 0,Y 369.4,Z 404.202,A -85,B 0,C 180,E1 -12548.738,E2 -12548.738} C_VEL
LIN {X 0,Y 369.04,Z 409.393,A -85,B 0,C 180,E1 -12549.618,E2 -12549.618} C_VEL
LIN {X 0,Y 368.71,Z 415.004,A -85,B 0,C 180,E1 -12550.755,E2 -12550.755} C_VEL
LIN {X 0,Y 368.299,Z 419.732,A -85,B 0,C 180,E1 -12551.911,E2 -12551.911} C_VEL
LIN {X 0,Y 368.091,Z 423.667,A -85,B 0,C 180,E1 -12553.09,E2 -12553.09} C_VEL
LIN {X 0,Y 367.888,Z 426.783,A -85,B 0,C 180,E1 -12554.246,E2 -12554.246} C_VEL
LIN {X 0,Y 367.631,Z 429.78,A -85,B 0,C 180,E1 -12555.753,E2 -12555.753} C_VEL
LIN {X 0,Y 367.542,Z 431.079,A -85,B 0,C 180,E1 -12556.602,E2 -12556.602} C_VEL
LIN {X 0,Y 367.42,Z 432.559,A -85,B 0,C 180,E1 -12558.243,E2 -12558.243} C_VEL
LIN {X 0,Y 367.48,Z 432.858,A -85,B 0,C 180,E1 -12559.905,E2 -12559.905} C_VEL
LIN {X 0,Y 367.551,Z 432.58,A -85,B 0,C 180,E1 -12560.878,E2 -12560.878} C_VEL
LIN {X 0,Y 367.725,Z 431.353,A -85,B 0,C 180,E1 -12562.297,E2 -12562.297} C_VEL
LIN {X 0,Y 367.996,Z 429.264,A -85,B 0,C 180,E1 -12563.7,E2 -12563.7} C_VEL
LIN {X 0,Y 368.355,Z 426.176,A -85,B 0,C 180,E1 -12565.124,E2 -12565.124} C_VEL
LIN {X 0,Y 368.895,Z 420.618,A -85,B 0,C 180,E1 -12566.955,E2 -12566.955} C_VEL
LIN {X 0,Y 369.425,Z 415.031,A -85,B 0,C 180,E1 -12568.358,E2 -12568.358} C_VEL
LIN {X 0,Y 370.103,Z 407.757,A -85,B 0,C 180,E1 -12569.788,E2 -12569.788} C_VEL
LIN {X 0,Y 370.87,Z 400.138,A -85,B 0,C 180,E1 -12570.958,E2 -12570.958} C_VEL
LIN {X 0,Y 371.536,Z 392.72,A -85,B 0,C 180,E1 -12571.893,E2 -12571.893} C_VEL
LIN {X 0,Y 372.074,Z 384.596,A -85,B 0,C 180,E1 -12572.733,E2 -12572.733} C_VEL
LIN {X 0,Y 372.563,Z 375.803,A -85,B 0,C 180,E1 -12573.46,E2 -12573.46} C_VEL
LIN {X 0,Y 373.141,Z 365.509,A -85,B 0,C 180,E1 -12574.106,E2 -12574.106} C_VEL
LIN {X 0,Y 373.495,Z 353.413,A -85,B 0,C 180,E1 -12574.618,E2 -12574.618} C_VEL
LIN {X 0,Y 373.855,Z 332.686,A -85,B 0,C 180,E1 -12575.105,E2 -12575.105} C_VEL
LIN {X 0,Y 374.573,Z 291.475,A -85,B 0,C 180,E1 -12575.996,E2 -12575.996} C_VEL
LIN {X 0,Y 371.975,Z 279.734,A -85,B 0,C 180,E1 -12576.417,E2 -12576.417} C_VEL
LIN {X 0,Y 369.923,Z 274.001,A -85,B 0,C 180,E1 -12576.71,E2 -12576.71} C_VEL
LIN {X 0,Y 368.92,Z 269.348,A -85,B 0,C 180,E1 -12577.974,E2 -12577.974} C_VEL
LIN {X 0,Y 368.972,Z 269.342,A -85,B 0,C 180,E1 -12581.108,E2 -12581.108} C_VEL
LIN {X 0,Y 368.987,Z 269.336,A -85,B 0,C 180,E1 -12584.536,E2 -12584.536} C_VEL
LIN {X 0,Y 368.996,Z 269.333,A -85,B 0,C 180,E1 -12587.907,E2 -12587.907} C_VEL
LIN {X 0,Y 369.157,Z 269.315,A -85,B 0,C 180,E1 -12591.87,E2 -12591.87} C_VEL
LIN {X 0,Y 369.139,Z 269.315,A -85,B 0,C 180,E1 -12594.538,E2 -12594.538} C_VEL
LIN {X 0,Y 369.31,Z 269.29,A -85,B 0,C 180,E1 -12597.82,E2 -12597.82} C_VEL
LIN {X 0,Y 369.449,Z 269.277,A -85,B 0,C 180,E1 -12600.001,E2 -12600.001} C_VEL
LIN {X 0,Y 369.311,Z 269.293,A -85,B 0,C 180,E1 -12602.182,E2 -12602.182} C_VEL
LIN {X 0,Y 369.2,Z 269.31,A -85,B 0,C 180,E1 -12606.559,E2 -12606.559} C_VEL
LIN {X 0,Y 369.13,Z 269.313,A -85,B 0,C 180,E1 -12608.762,E2 -12608.762} C_VEL
LIN {X 0,Y 368.997,Z 269.329,A -85,B 0,C 180,E1 -12612.094,E2 -12612.094} C_VEL
LIN {X 0,Y 368.991,Z 269.331,A -85,B 0,C 180,E1 -12615.466,E2 -12615.466} C_VEL
LIN {X 0,Y 368.976,Z 269.335,A -85,B 0,C 180,E1 -12618.894,E2 -12618.894} C_VEL
LIN {X 0,Y 368.926,Z 269.34,A -85,B 0,C 180,E1 -12622.396,E2 -12622.396} C_VEL
LIN {X 0,Y 368.994,Z 269.326,A -85,B 0,C 180,E1 -12625.981,E2 -12625.981} C_VEL
LIN {X 0,Y 368.962,Z 269.331,A -85,B 0,C 180,E1 -12628.814,E2 -12628.814} C_VEL
LIN {X 0,Y 368.895,Z 269.348,A -85,B 0,C 180,E1 -12632.239,E2 -12632.239} C_VEL
LIN {X 0,Y 368.925,Z 269.342,A -85,B 0,C 180,E1 -12635.003,E2 -12635.003} C_VEL
LIN {X 0,Y 368.91,Z 269.347,A -85,B 0,C 180,E1 -12638.642,E2 -12638.642} C_VEL
LIN {X 0,Y 368.907,Z 269.343,A -85,B 0,C 180,E1 -12641.82,E2 -12641.82} C_VEL
LIN {X 0,Y 368.881,Z 269.347,A -85,B 0,C 180,E1 -12645.178,E2 -12645.178} C_VEL
LIN {X 0,Y 368.881,Z 269.35,A -85,B 0,C 180,E1 -12648.179,E2 -12648.179} C_VEL
LIN {X 0,Y 368.908,Z 269.343,A -85,B 0,C 180,E1 -12651.361,E2 -12651.361} C_VEL
LIN {X 0,Y 368.936,Z 269.341,A -85,B 0,C 180,E1 -12655.148,E2 -12655.148} C_VEL
LIN {X 0,Y 368.929,Z 269.344,A -85,B 0,C 180,E1 -12659.047,E2 -12659.047} C_VEL
LIN {X 0,Y 368.979,Z 269.419,A -85,B 0,C 180,E1 -12662.53,E2 -12662.53} C_VEL
LIN {X 0,Y 370.964,Z 279.317,A -85,B 0,C 180,E1 -12665.07,E2 -12665.07} C_VEL
LIN {X 0,Y 371.337,Z 284.343,A -85,B 0,C 180,E1 -12666.286,E2 -12666.286} C_VEL
LIN {X 0,Y 370.111,Z 300.567,A -85,B 0,C 180,E1 -12670.014,E2 -12670.014} C_VEL
LIN {X 0,Y 369.498,Z 310.817,A -85,B 0,C 180,E1 -12672.346,E2 -12672.346} C_VEL
LIN {X 0,Y 372.781,Z 331.96,A -85,B 0,C 180,E1 -12673.019,E2 -12673.019} C_VEL
LIN {X 0,Y 373.924,Z 344.783,A -85,B 0,C 180,E1 -12673.372,E2 -12673.372} C_VEL
LIN {X 0,Y 373.038,Z 390.343,A -85,B 0,C 180,E1 -12674.373,E2 -12674.373} C_VEL
LIN {X 0,Y 372.547,Z 402.259,A -85,B 0,C 180,E1 -12674.827,E2 -12674.827} C_VEL
LIN {X 0,Y 371.787,Z 413.489,A -85,B 0,C 180,E1 -12675.495,E2 -12675.495} C_VEL
LIN {X 0,Y 371.093,Z 422.085,A -85,B 0,C 180,E1 -12676.167,E2 -12676.167} C_VEL
LIN {X 0,Y 370.394,Z 430.366,A -85,B 0,C 180,E1 -12676.979,E2 -12676.979} C_VEL
LIN {X 0,Y 369.64,Z 438.254,A -85,B 0,C 180,E1 -12677.928,E2 -12677.928} C_VEL
LIN {X 0,Y 369.066,Z 445.666,A -85,B 0,C 180,E1 -12679.023,E2 -12679.023} C_VEL
LIN {X 0,Y 368.405,Z 453.201,A -85,B 0,C 180,E1 -12680.392,E2 -12680.392} C_VEL
LIN {X 0,Y 367.957,Z 459.109,A -85,B 0,C 180,E1 -12681.764,E2 -12681.764} C_VEL
LIN {X 0,Y 367.748,Z 463.006,A -85,B 0,C 180,E1 -12682.865,E2 -12682.865} C_VEL
LIN {X 0,Y 367.498,Z 467.464,A -85,B 0,C 180,E1 -12684.513,E2 -12684.513} C_VEL
LIN {X 0,Y 367.545,Z 469.765,A -85,B 0,C 180,E1 -12685.614,E2 -12685.614} C_VEL
LIN {X 0,Y 367.459,Z 471.471,A -85,B 0,C 180,E1 -12686.711,E2 -12686.711} C_VEL
LIN {X 0,Y 367.525,Z 472.576,A -85,B 0,C 180,E1 -12687.809,E2 -12687.809} C_VEL
LIN {X 0,Y 367.579,Z 473.186,A -85,B 0,C 180,E1 -12688.905,E2 -12688.905} C_VEL
LIN {X 0,Y 367.582,Z 473.312,A -85,B 0,C 180,E1 -12690,E2 -12690} C_VEL
LIN {X 0,Y 367.588,Z 472.951,A -85,B 0,C 180,E1 -12691.096,E2 -12691.096} C_VEL
LIN {X 0,Y 367.568,Z 472.004,A -85,B 0,C 180,E1 -12692.192,E2 -12692.192} C_VEL
LIN {X 0,Y 367.508,Z 469.578,A -85,B 0,C 180,E1 -12693.838,E2 -12693.838} C_VEL
LIN {X 0,Y 367.565,Z 467.246,A -85,B 0,C 180,E1 -12694.936,E2 -12694.936} C_VEL
LIN {X 0,Y 367.644,Z 462.5,A -85,B 0,C 180,E1 -12696.586,E2 -12696.586} C_VEL
LIN {X 0,Y 367.87,Z 457.309,A -85,B 0,C 180,E1 -12697.962,E2 -12697.962} C_VEL
LIN {X 0,Y 368.152,Z 452.225,A -85,B 0,C 180,E1 -12699.061,E2 -12699.061} C_VEL
LIN {X 0,Y 368.52,Z 446.09,A -85,B 0,C 180,E1 -12700.161,E2 -12700.161} C_VEL
LIN {X 0,Y 368.953,Z 439.655,A -85,B 0,C 180,E1 -12701.12,E2 -12701.12} C_VEL
